// TIA Portal V16 export
// export: Created 2021-11-12T13:31:15.9471578Z, ExportSetting WithDefaults, DisplayName Totally Integrated Automation Portal, DisplayVersion V16 Update 3, DisplayName TIA Portal Version Control Interface, DisplayVersion V16 Update 2, DisplayName TIA Portal Openness, DisplayVersion V16 Update 3, DisplayName SINAMICS Startdrive Advanced, DisplayVersion V16 Update 5, DisplayName SINAMICS Startdrive G130, G150, S120, S150, SINAMICS MV, S210, DisplayVersion V16 Update 5, DisplayName SINAMICS Startdrive G110M, G120, G120C, G120D, G120P, G115D, DisplayVersion V16 Update 5, DisplayName STEP 7 Professional, DisplayVersion V16 Update 3, DisplayName STEP 7 Safety, DisplayVersion V16, DisplayName WinCC UA Professional, DisplayVersion V16 Update 3
FUNCTION_BLOCK "STD_RobotABB"   // FB1225, LAD
TITLE = STD_RobotABB
{ S7_Optimized_Access := 'TRUE' }
VERSION : 0.1
// Robot control
// stored: AutoNumber false, IsIECCheckEnabled false, IsRetainMemResEnabled false, MemoryReserve 100, SetENOAutomatically false, UDAEnableTagReadback false
   VAR_INPUT
      IS_ZoneM { ExternalAccessible := 'False'; ExternalVisible := 'False'; ExternalWritable := 'False'} : "UDT_Status_main";   // Main structure from zone
      IS_ZoneS { ExternalAccessible := 'False'; ExternalVisible := 'False'; ExternalWritable := 'False'} : "UDT_Zone_Status_specific";   // Specific structure from zone
      IS_Robot : "UDT_RobotABB_RobotDI";
      IS_Intl : "UDT_RobotABB_Interlock";
      IS_ZoneRel : "UDT_RobotABB_ZoneReleaseToRobot";
      IB1CtrlRun : Bool;   // Controller running in auto mode
      IB1LimSpd : Bool;   // Set robot maximal speed to safe speed (250mm/s default)
      IB1CnclJob : Bool;   // Cancel of robot job
      IB1StartJob : Bool;   // Start robot job - job number valid
      IB1AckEndOfJob : Bool;   // Acknowledge end of robot job
      IB1AlmSupp : Bool;   // Suppress alarms
      II_JobNr : UInt;   // Robot job number
      II_TypeNr : UInt;   // Robot type number
      II_PosNr : UInt;   // Robot position specification
   END_VAR
   VAR_OUTPUT
      OS_Status : Struct
         Main : "UDT_Status_main";
         Specific : "UDT_RobotABB_Status_specific";
         Error : "UDT_Error01";
      END_STRUCT;
      OS_Robot : "UDT_RobotABB_RobotDO";
   END_VAR
   VAR_IN_OUT
      XS_Parameter : "UDT_RobotABB_Parameter";
      XS_Command : "UDT_RobotABB_Command";
   END_VAR
   VAR
      SS_Alarm : Struct   // Device alarms
         RobotErr : Bool;   // Robot error - See teachpendant for further information
         Colsn : Bool;   // Motion supervision triggered
         JobNrNotMatch : Bool;   // Job number feedback does not match
         TypeNrNotMatch : Bool;   // Type number feedback does not match
         Res_0_4 : Bool;   // Reserve
         Res_0_5 : Bool;   // Reserve
         Res_0_6 : Bool;   // Reserve
         Res_0_7 : Bool;   // Reserve
      END_STRUCT;
      SS_Warning : Struct   // Device warnings
         LimSpd : Bool;   // Speed is limited to safe speed (250mm/s by default)
         NoTaskExec : Bool;   // Robot is not executing task
         NotOnPath : Bool;   // Robot is not on programmed path
         Res_0_3 : Bool;   // Reserve
         Res_0_4 : Bool;   // Reserve
         Res_0_5 : Bool;   // Reserve
         Res_0_6 : Bool;   // Reserve
         Res_0_7 : Bool;   // Reserve
      END_STRUCT;
      SS_RobotIn { S7_SetPoint := 'True'} : "UDT_RobotABB_RobotDI";
      SS_RobotOut { S7_SetPoint := 'True'} : "UDT_RobotABB_RobotDO";
      SS_SeqNr : UInt;
      SB1CollErr : Bool;   // Collective error from device
      SB1CollWrn : Bool;   // Collective warning from device
      SB1RobotReady : Bool;   // Robot ready to operation
      SB1StartJobReq : Bool;   // Start job request is detected
      SB1InitReq : Bool;   // Robot init request
      SB1InitTrg : Bool;   // Robot init request trigger
      SB1TrigPE1 : Bool;
      SB1TrigPE2 : Bool;
      SB1TrigPE3 : Bool;
      SB1CnclJobPE : Bool;
      SB1ServicePosReq : Bool;   // Request to go to/from service position
   END_VAR
   VAR_TEMP
      TS_Status : Struct
         Main : "UDT_Status_main";
         Specific : "UDT_RobotABB_Status_specific";
         Error : "UDT_Error01";
      END_STRUCT;
      TS_Parameter : "UDT_RobotABB_Parameter";
      TS_ZoneRel : Struct
         Zone : Array[0..#CI_StnNr] of Struct
            Allowed : Bool;
         END_STRUCT;
      END_STRUCT;
      TS_Intl : Struct
         Station : Array[0..#CI_StnNr] of Word;
      END_STRUCT;
      TS_Command : "UDT_RobotABB_Command";
      TW_StnIntlSpec : Word;
      "TW _StnIntlMask" : Word;   // Interlocks condition masked by request
      TW_StnIntlAckSpec : Word;   // Interlock conditions fulfilled PLC->Robot (selected station only)
      TI_StnIntlSpec : UInt;   // Interlock request Robot->PLC (Nr. of interlock in specific station)
      TI_IntStnNr : UInt;   // Interlock request Robot->PLC (station number)
      TI_RobotIntlAdj : UInt;   // Interlock number adjusted
      TI_InterlockLim : UInt;   // Interlock limitation
      TB1AckPulse : Bool;
      TB1AlmSupp : Bool;
      TI_RetVal : Int;
   END_VAR
   VAR CONSTANT
      CI_StnNr : UInt := 8;   // Number of stations used in Interfaces
   END_VAR
   VAR_TEMP   // added for the SCL form of the ladder/FBD networks
      _w1 : Bool;
      _w2 : Bool;
      _w3 : Bool;
      _w4 : Bool;
      _w5 : Bool;
   END_VAR
BEGIN

REGION Network 1: Clear temporary TS_Status - Main, Specific
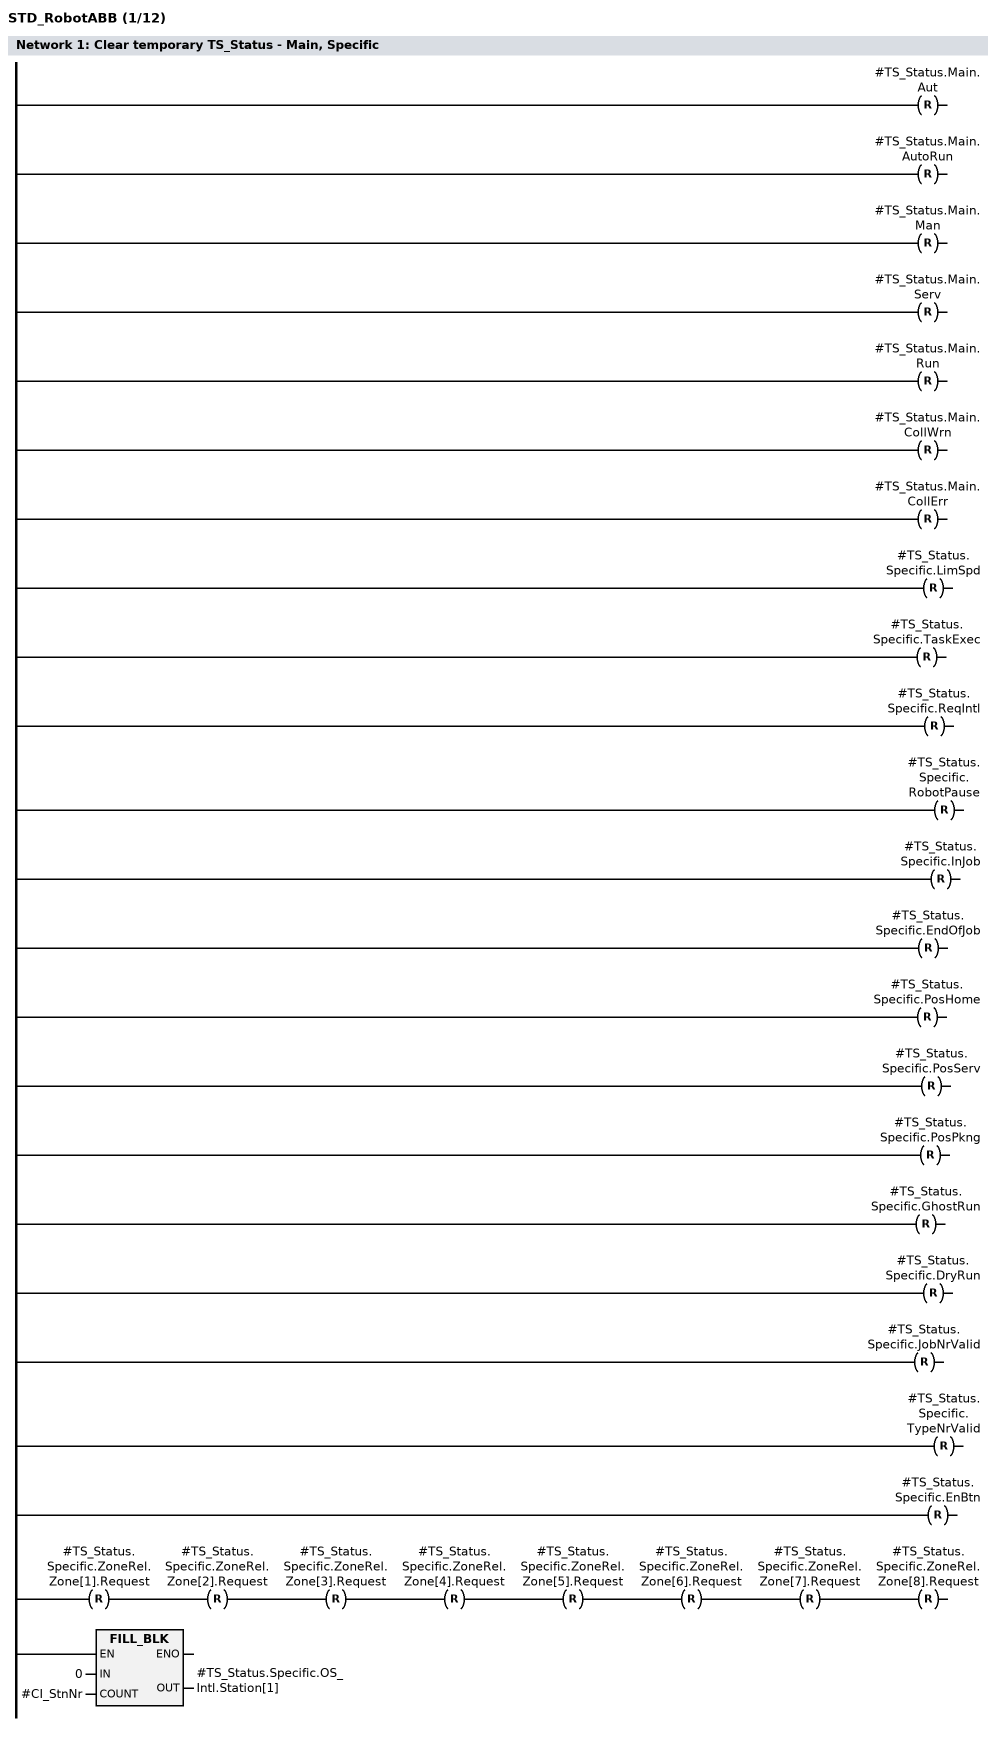
   RUNG wire#powerrail
      R_Coil( #TS_Status.Main.Aut )
   END_RUNG
   RUNG wire#powerrail
      R_Coil( #TS_Status.Main.AutoRun )
   END_RUNG
   RUNG wire#powerrail
      R_Coil( #TS_Status.Main.Man )
   END_RUNG
   RUNG wire#powerrail
      R_Coil( #TS_Status.Main.Serv )
   END_RUNG
   RUNG wire#powerrail
      R_Coil( #TS_Status.Main.Run )
   END_RUNG
   RUNG wire#powerrail
      R_Coil( #TS_Status.Main.CollWrn )
   END_RUNG
   RUNG wire#powerrail
      R_Coil( #TS_Status.Main.CollErr )
   END_RUNG
   RUNG wire#powerrail
      R_Coil( #TS_Status.Specific.LimSpd )
   END_RUNG
   RUNG wire#powerrail
      R_Coil( #TS_Status.Specific.TaskExec )
   END_RUNG
   RUNG wire#powerrail
      R_Coil( #TS_Status.Specific.ReqIntl )
   END_RUNG
   RUNG wire#powerrail
      R_Coil( #TS_Status.Specific.RobotPause )
   END_RUNG
   RUNG wire#powerrail
      R_Coil( #TS_Status.Specific.InJob )
   END_RUNG
   RUNG wire#powerrail
      R_Coil( #TS_Status.Specific.EndOfJob )
   END_RUNG
   RUNG wire#powerrail
      R_Coil( #TS_Status.Specific.PosHome )
   END_RUNG
   RUNG wire#powerrail
      R_Coil( #TS_Status.Specific.PosServ )
   END_RUNG
   RUNG wire#powerrail
      R_Coil( #TS_Status.Specific.PosPkng )
   END_RUNG
   RUNG wire#powerrail
      R_Coil( #TS_Status.Specific.GhostRun )
   END_RUNG
   RUNG wire#powerrail
      R_Coil( #TS_Status.Specific.DryRun )
   END_RUNG
   RUNG wire#powerrail
      R_Coil( #TS_Status.Specific.JobNrValid )
   END_RUNG
   RUNG wire#powerrail
      R_Coil( #TS_Status.Specific.TypeNrValid )
   END_RUNG
   RUNG wire#powerrail
      R_Coil( #TS_Status.Specific.EnBtn )
   END_RUNG
   RUNG wire#powerrail
      R_Coil( #TS_Status.Specific.ZoneRel.Zone[1].Request )
      R_Coil( #TS_Status.Specific.ZoneRel.Zone[2].Request )
      R_Coil( #TS_Status.Specific.ZoneRel.Zone[3].Request )
      R_Coil( #TS_Status.Specific.ZoneRel.Zone[4].Request )
      R_Coil( #TS_Status.Specific.ZoneRel.Zone[5].Request )
      R_Coil( #TS_Status.Specific.ZoneRel.Zone[6].Request )
      R_Coil( #TS_Status.Specific.ZoneRel.Zone[7].Request )
      R_Coil( #TS_Status.Specific.ZoneRel.Zone[8].Request )
   END_RUNG
   RUNG wire#powerrail
      { S7_GenerateENO := "TRUE" } FillBlockI(in := 0, count := #CI_StnNr, out => #TS_Status.Specific.OS_Intl.Station[1])
   END_RUNG
   // the same network as SCL:
   #TS_Status.Main.Aut := FALSE;
   #TS_Status.Main.AutoRun := FALSE;
   #TS_Status.Main.Man := FALSE;
   #TS_Status.Main.Serv := FALSE;
   #TS_Status.Main.Run := FALSE;
   #TS_Status.Main.CollWrn := FALSE;
   #TS_Status.Main.CollErr := FALSE;
   #TS_Status.Specific.LimSpd := FALSE;
   #TS_Status.Specific.TaskExec := FALSE;
   #TS_Status.Specific.ReqIntl := FALSE;
   #TS_Status.Specific.RobotPause := FALSE;
   #TS_Status.Specific.InJob := FALSE;
   #TS_Status.Specific.EndOfJob := FALSE;
   #TS_Status.Specific.PosHome := FALSE;
   #TS_Status.Specific.PosServ := FALSE;
   #TS_Status.Specific.PosPkng := FALSE;
   #TS_Status.Specific.GhostRun := FALSE;
   #TS_Status.Specific.DryRun := FALSE;
   #TS_Status.Specific.JobNrValid := FALSE;
   #TS_Status.Specific.TypeNrValid := FALSE;
   #TS_Status.Specific.EnBtn := FALSE;
   #TS_Status.Specific.ZoneRel.Zone[1].Request := FALSE;
   #TS_Status.Specific.ZoneRel.Zone[2].Request := FALSE;
   #TS_Status.Specific.ZoneRel.Zone[3].Request := FALSE;
   #TS_Status.Specific.ZoneRel.Zone[4].Request := FALSE;
   #TS_Status.Specific.ZoneRel.Zone[5].Request := FALSE;
   #TS_Status.Specific.ZoneRel.Zone[6].Request := FALSE;
   #TS_Status.Specific.ZoneRel.Zone[7].Request := FALSE;
   #TS_Status.Specific.ZoneRel.Zone[8].Request := FALSE;
   FILL_BLK(IN := 0, COUNT := #CI_StnNr, OUT => #TS_Status.Specific.OS_Intl.Station[1]);
END_REGION

REGION Network 2: Copy In/Out variables to temporary variables
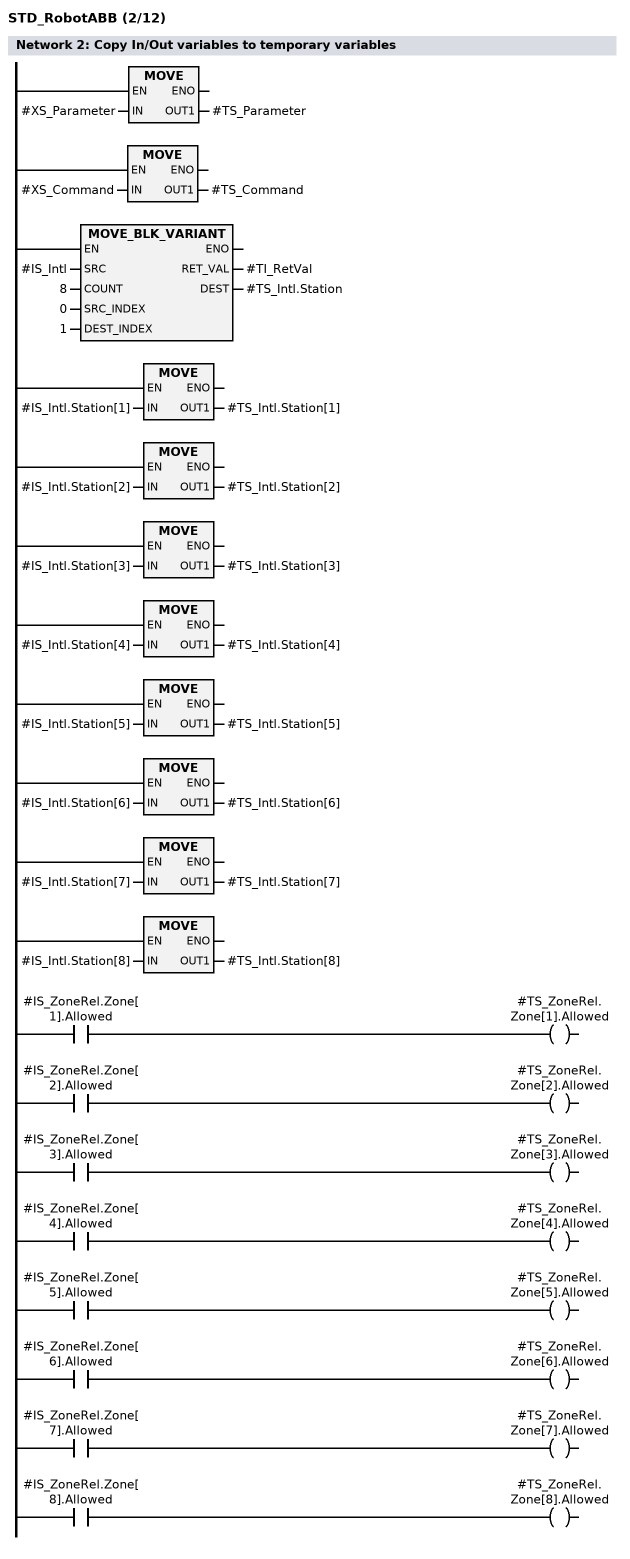
   RUNG wire#powerrail
      { S7_GenerateENO := "TRUE" } Move(in := #XS_Parameter, out1 => #TS_Parameter)
   END_RUNG
   RUNG wire#powerrail
      { S7_GenerateENO := "TRUE" } Move(in := #XS_Command, out1 => #TS_Command)
   END_RUNG
   RUNG wire#powerrail
      MOVE_BLK_VARIANT(SRC := #IS_Intl, COUNT := 8, SRC_INDEX := 0, DEST_INDEX := 1, Ret_Val => #TI_RetVal, DEST => #TS_Intl.Station)
   END_RUNG
   RUNG wire#powerrail
      Move(in := #IS_Intl.Station[1], out1 => #TS_Intl.Station[1])
   END_RUNG
   RUNG wire#powerrail
      Move(in := #IS_Intl.Station[2], out1 => #TS_Intl.Station[2])
   END_RUNG
   RUNG wire#powerrail
      Move(in := #IS_Intl.Station[3], out1 => #TS_Intl.Station[3])
   END_RUNG
   RUNG wire#powerrail
      Move(in := #IS_Intl.Station[4], out1 => #TS_Intl.Station[4])
   END_RUNG
   RUNG wire#powerrail
      Move(in := #IS_Intl.Station[5], out1 => #TS_Intl.Station[5])
   END_RUNG
   RUNG wire#powerrail
      Move(in := #IS_Intl.Station[6], out1 => #TS_Intl.Station[6])
   END_RUNG
   RUNG wire#powerrail
      Move(in := #IS_Intl.Station[7], out1 => #TS_Intl.Station[7])
   END_RUNG
   RUNG wire#powerrail
      Move(in := #IS_Intl.Station[8], out1 => #TS_Intl.Station[8])
   END_RUNG
   RUNG wire#powerrail
      Contact( #IS_ZoneRel.Zone[1].Allowed )
      Coil( #TS_ZoneRel.Zone[1].Allowed )
   END_RUNG
   RUNG wire#powerrail
      Contact( #IS_ZoneRel.Zone[2].Allowed )
      Coil( #TS_ZoneRel.Zone[2].Allowed )
   END_RUNG
   RUNG wire#powerrail
      Contact( #IS_ZoneRel.Zone[3].Allowed )
      Coil( #TS_ZoneRel.Zone[3].Allowed )
   END_RUNG
   RUNG wire#powerrail
      Contact( #IS_ZoneRel.Zone[4].Allowed )
      Coil( #TS_ZoneRel.Zone[4].Allowed )
   END_RUNG
   RUNG wire#powerrail
      Contact( #IS_ZoneRel.Zone[5].Allowed )
      Coil( #TS_ZoneRel.Zone[5].Allowed )
   END_RUNG
   RUNG wire#powerrail
      Contact( #IS_ZoneRel.Zone[6].Allowed )
      Coil( #TS_ZoneRel.Zone[6].Allowed )
   END_RUNG
   RUNG wire#powerrail
      Contact( #IS_ZoneRel.Zone[7].Allowed )
      Coil( #TS_ZoneRel.Zone[7].Allowed )
   END_RUNG
   RUNG wire#powerrail
      Contact( #IS_ZoneRel.Zone[8].Allowed )
      Coil( #TS_ZoneRel.Zone[8].Allowed )
   END_RUNG
   // the same network as SCL:
   #TS_Parameter := #XS_Parameter;
   #TS_Command := #XS_Command;
   #TI_RetVal := MOVE_BLK_VARIANT(SRC := #IS_Intl,
                           COUNT := 8,
                           SRC_INDEX := 0,
                           DEST_INDEX := 1,
                           DEST => #TS_Intl.Station);
   #TS_Intl.Station[1] := #IS_Intl.Station[1];
   #TS_Intl.Station[2] := #IS_Intl.Station[2];
   #TS_Intl.Station[3] := #IS_Intl.Station[3];
   #TS_Intl.Station[4] := #IS_Intl.Station[4];
   #TS_Intl.Station[5] := #IS_Intl.Station[5];
   #TS_Intl.Station[6] := #IS_Intl.Station[6];
   #TS_Intl.Station[7] := #IS_Intl.Station[7];
   #TS_Intl.Station[8] := #IS_Intl.Station[8];
   #TS_ZoneRel.Zone[1].Allowed := #IS_ZoneRel.Zone[1].Allowed;
   #TS_ZoneRel.Zone[2].Allowed := #IS_ZoneRel.Zone[2].Allowed;
   #TS_ZoneRel.Zone[3].Allowed := #IS_ZoneRel.Zone[3].Allowed;
   #TS_ZoneRel.Zone[4].Allowed := #IS_ZoneRel.Zone[4].Allowed;
   #TS_ZoneRel.Zone[5].Allowed := #IS_ZoneRel.Zone[5].Allowed;
   #TS_ZoneRel.Zone[6].Allowed := #IS_ZoneRel.Zone[6].Allowed;
   #TS_ZoneRel.Zone[7].Allowed := #IS_ZoneRel.Zone[7].Allowed;
   #TS_ZoneRel.Zone[8].Allowed := #IS_ZoneRel.Zone[8].Allowed;
END_REGION

REGION Network 3: Merge of alarm suppress
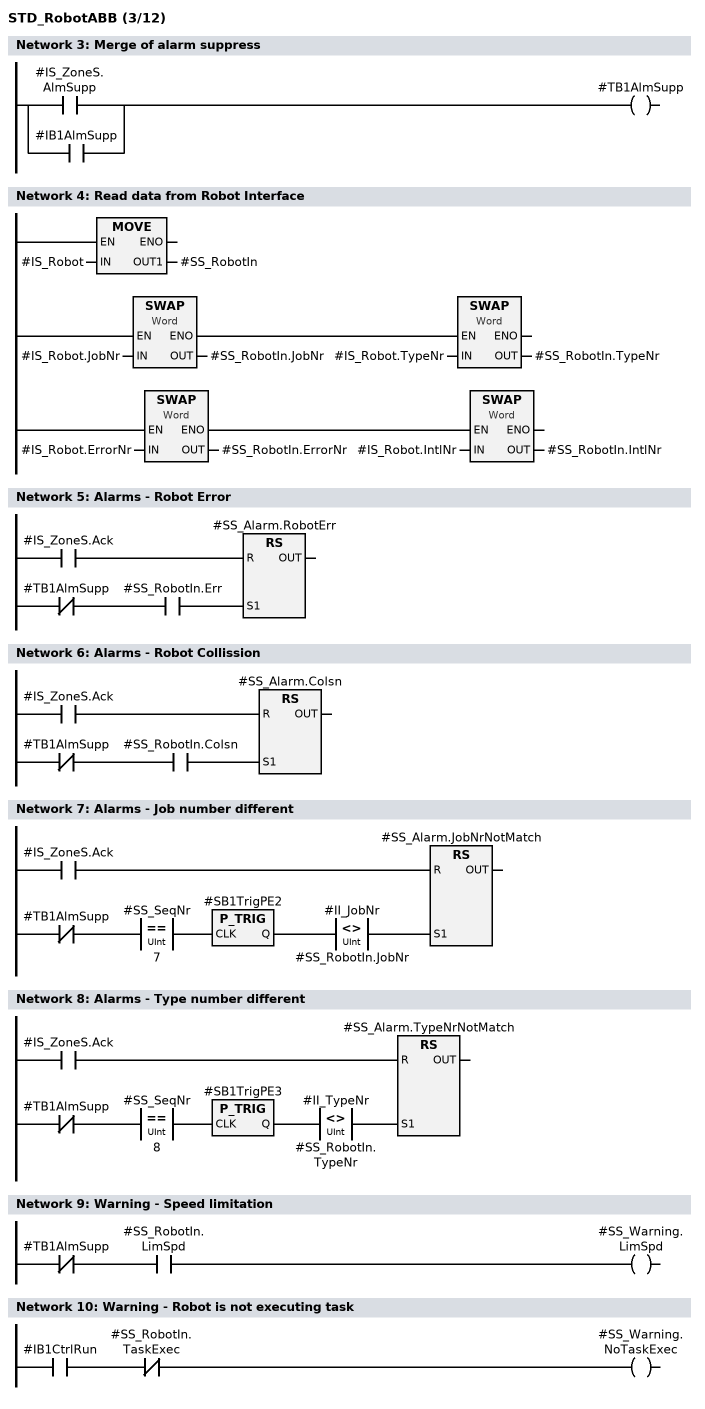
   RUNG wire#powerrail
      Contact( #IS_ZoneS.AlmSupp )
      wire#w1
      Coil( #TB1AlmSupp )
   END_RUNG
   RUNG wire#powerrail
      Contact( #IB1AlmSupp )
   END_RUNG wire#w1
   // the same network as SCL:
   #TB1AlmSupp := #IS_ZoneS.AlmSupp OR #IB1AlmSupp;
END_REGION

REGION Network 4: Read data from Robot Interface
   #SS_RobotIn := #IS_Robot;
   #SS_RobotIn.JobNr := SWAP(#IS_Robot.JobNr);
   #SS_RobotIn.TypeNr := SWAP(#IS_Robot.TypeNr);
   #SS_RobotIn.ErrorNr := SWAP(#IS_Robot.ErrorNr);
   #SS_RobotIn.IntlNr := SWAP(#IS_Robot.IntlNr);
END_REGION

REGION Network 5: Alarms - Robot Error
   RUNG wire#powerrail
      Contact( #IS_ZoneS.Ack )
      S_RS(operand := #SS_Alarm.RobotErr, s1 := wire#w1)
   END_RUNG
   RUNG wire#powerrail
      I_Contact( #TB1AlmSupp )
      Contact( #SS_RobotIn.Err )
   END_RUNG wire#w1
   // the same network as SCL:
   IF #IS_ZoneS.Ack THEN
       #SS_Alarm.RobotErr := FALSE;   // RS flip-flop
   END_IF;
   IF NOT #TB1AlmSupp AND #SS_RobotIn.Err THEN #SS_Alarm.RobotErr := TRUE; END_IF;
END_REGION

REGION Network 6: Alarms - Robot Collission
   RUNG wire#powerrail
      Contact( #IS_ZoneS.Ack )
      S_RS(operand := #SS_Alarm.Colsn, s1 := wire#w1)
   END_RUNG
   RUNG wire#powerrail
      I_Contact( #TB1AlmSupp )
      Contact( #SS_RobotIn.Colsn )
   END_RUNG wire#w1
   // the same network as SCL:
   IF #IS_ZoneS.Ack THEN
       #SS_Alarm.Colsn := FALSE;   // RS flip-flop
   END_IF;
   IF NOT #TB1AlmSupp AND #SS_RobotIn.Colsn THEN #SS_Alarm.Colsn := TRUE; END_IF;
END_REGION

REGION Network 7: Alarms - Job number different
   RUNG wire#powerrail
      Contact( #IS_ZoneS.Ack )
      S_RS(operand := #SS_Alarm.JobNrNotMatch, s1 := wire#w1)
   END_RUNG
   RUNG wire#powerrail
      I_Contact( #TB1AlmSupp )
      { S7_Templates := "SrcType := UInt" } EQ_Contact(in1 := #SS_SeqNr, in2 := 7)
      P_Trig( #SB1TrigPE2 )
      { S7_Templates := "SrcType := UInt" } NE_Contact(in1 := #II_JobNr, in2 := #SS_RobotIn.JobNr)
   END_RUNG wire#w1
   // the same network as SCL:
   #_w1 := NOT #TB1AlmSupp AND (#SS_SeqNr = 7);
   #_w2 := #_w1 AND NOT #SB1TrigPE2;   // rising edge
   #SB1TrigPE2 := #_w1;
   IF #IS_ZoneS.Ack THEN
       #SS_Alarm.JobNrNotMatch := FALSE;   // RS flip-flop
   END_IF;
   IF #_w2 AND (#II_JobNr <> #SS_RobotIn.JobNr) THEN #SS_Alarm.JobNrNotMatch := TRUE; END_IF;
END_REGION

REGION Network 8: Alarms - Type number different
   RUNG wire#powerrail
      Contact( #IS_ZoneS.Ack )
      S_RS(operand := #SS_Alarm.TypeNrNotMatch, s1 := wire#w1)
   END_RUNG
   RUNG wire#powerrail
      I_Contact( #TB1AlmSupp )
      { S7_Templates := "SrcType := UInt" } EQ_Contact(in1 := #SS_SeqNr, in2 := 8)
      P_Trig( #SB1TrigPE3 )
      { S7_Templates := "SrcType := UInt" } NE_Contact(in1 := #II_TypeNr, in2 := #SS_RobotIn.TypeNr)
   END_RUNG wire#w1
   // the same network as SCL:
   #_w1 := NOT #TB1AlmSupp AND (#SS_SeqNr = 8);
   #_w2 := #_w1 AND NOT #SB1TrigPE3;   // rising edge
   #SB1TrigPE3 := #_w1;
   IF #IS_ZoneS.Ack THEN
       #SS_Alarm.TypeNrNotMatch := FALSE;   // RS flip-flop
   END_IF;
   IF #_w2 AND (#II_TypeNr <> #SS_RobotIn.TypeNr) THEN #SS_Alarm.TypeNrNotMatch := TRUE; END_IF;
END_REGION

REGION Network 9: Warning - Speed limitation
   RUNG wire#powerrail
      I_Contact( #TB1AlmSupp )
      Contact( #SS_RobotIn.LimSpd )
      Coil( #SS_Warning.LimSpd )
   END_RUNG
   // the same network as SCL:
   #SS_Warning.LimSpd := NOT #TB1AlmSupp AND #SS_RobotIn.LimSpd;
END_REGION

REGION Network 10: Warning - Robot is not executing task
   RUNG wire#powerrail
      Contact( #IB1CtrlRun )
      I_Contact( #SS_RobotIn.TaskExec )
      Coil( #SS_Warning.NoTaskExec )
   END_RUNG
   // the same network as SCL:
   #SS_Warning.NoTaskExec := #IB1CtrlRun AND NOT #SS_RobotIn.TaskExec;
END_REGION

REGION Network 11: Warning - Robot is not programmed path
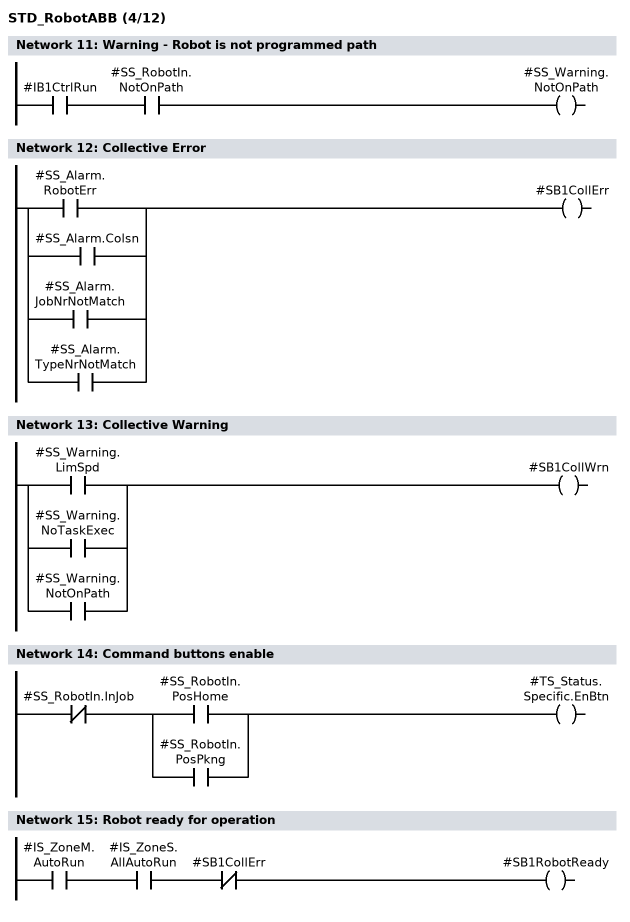
   RUNG wire#powerrail
      Contact( #IB1CtrlRun )
      Contact( #SS_RobotIn.NotOnPath )
      Coil( #SS_Warning.NotOnPath )
   END_RUNG
   // the same network as SCL:
   #SS_Warning.NotOnPath := #IB1CtrlRun AND #SS_RobotIn.NotOnPath;
END_REGION

REGION Network 12: Collective Error
   RUNG wire#powerrail
      Contact( #SS_Alarm.RobotErr )
      wire#w1
      Coil( #SB1CollErr )
   END_RUNG
   RUNG wire#powerrail
      Contact( #SS_Alarm.Colsn )
   END_RUNG wire#w1
   RUNG wire#powerrail
      Contact( #SS_Alarm.JobNrNotMatch )
   END_RUNG wire#w1
   RUNG wire#powerrail
      Contact( #SS_Alarm.TypeNrNotMatch )
   END_RUNG wire#w1
   // the same network as SCL:
   #SB1CollErr := #SS_Alarm.RobotErr OR #SS_Alarm.Colsn OR #SS_Alarm.JobNrNotMatch OR #SS_Alarm.TypeNrNotMatch;
END_REGION

REGION Network 13: Collective Warning
   RUNG wire#powerrail
      Contact( #SS_Warning.LimSpd )
      wire#w1
      Coil( #SB1CollWrn )
   END_RUNG
   RUNG wire#powerrail
      Contact( #SS_Warning.NoTaskExec )
   END_RUNG wire#w1
   RUNG wire#powerrail
      Contact( #SS_Warning.NotOnPath )
   END_RUNG wire#w1
   // the same network as SCL:
   #SB1CollWrn := #SS_Warning.LimSpd OR #SS_Warning.NoTaskExec OR #SS_Warning.NotOnPath;
END_REGION

REGION Network 14: Command buttons enable
   RUNG wire#powerrail
      I_Contact( #SS_RobotIn.InJob )
      wire#w1
      Contact( #SS_RobotIn.PosHome )
      wire#w2
      Coil( #TS_Status.Specific.EnBtn )
   END_RUNG
   RUNG wire#w1
      Contact( #SS_RobotIn.PosPkng )
   END_RUNG wire#w2
   // the same network as SCL:
   #TS_Status.Specific.EnBtn := NOT #SS_RobotIn.InJob AND (#SS_RobotIn.PosHome OR #SS_RobotIn.PosPkng);
END_REGION

REGION Network 15: Robot ready for operation
   RUNG wire#powerrail
      Contact( #IS_ZoneM.AutoRun )
      Contact( #IS_ZoneS.AllAutoRun )
      I_Contact( #SB1CollErr )
      Coil( #SB1RobotReady )
   END_RUNG
   // the same network as SCL:
   #SB1RobotReady := #IS_ZoneM.AutoRun AND #IS_ZoneS.AllAutoRun AND NOT #SB1CollErr;
END_REGION

REGION Network 16: Dry Run / Ghost Run
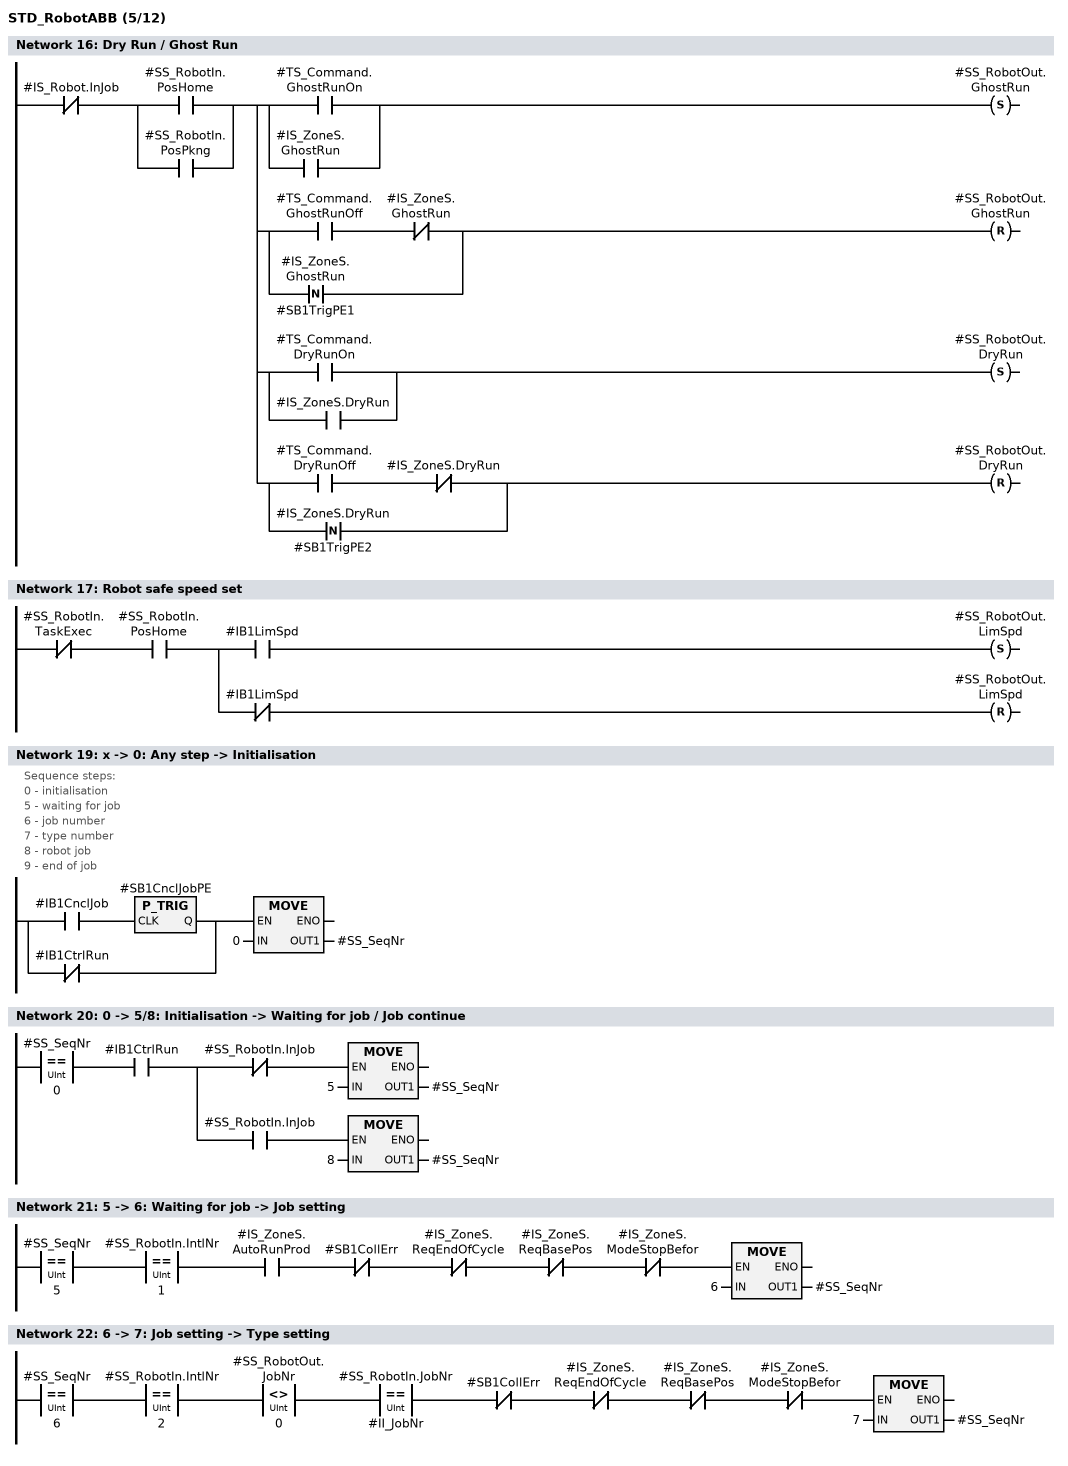
   RUNG wire#powerrail
      I_Contact( #IS_Robot.InJob )
      wire#w1
      Contact( #SS_RobotIn.PosHome )
      wire#w2
      Contact( #TS_Command.GhostRunOn )
      wire#w3
      S_Coil( #SS_RobotOut.GhostRun )
   END_RUNG
   RUNG wire#w1
      Contact( #SS_RobotIn.PosPkng )
   END_RUNG wire#w2
   RUNG wire#w2
      Contact( #IS_ZoneS.GhostRun )
   END_RUNG wire#w3
   RUNG wire#w2
      Contact( #TS_Command.GhostRunOff )
      I_Contact( #IS_ZoneS.GhostRun )
      wire#w4
      R_Coil( #SS_RobotOut.GhostRun )
   END_RUNG
   RUNG wire#w2
      N_Contact(operand := #IS_ZoneS.GhostRun, bit := #SB1TrigPE1)
   END_RUNG wire#w4
   RUNG wire#w2
      Contact( #TS_Command.DryRunOn )
      wire#w5
      S_Coil( #SS_RobotOut.DryRun )
   END_RUNG
   RUNG wire#w2
      Contact( #IS_ZoneS.DryRun )
   END_RUNG wire#w5
   RUNG wire#w2
      Contact( #TS_Command.DryRunOff )
      I_Contact( #IS_ZoneS.DryRun )
      wire#w6
      R_Coil( #SS_RobotOut.DryRun )
   END_RUNG
   RUNG wire#w2
      N_Contact(operand := #IS_ZoneS.DryRun, bit := #SB1TrigPE2)
   END_RUNG wire#w6
   // the same network as SCL:
   #_w1 := NOT #IS_Robot.InJob AND (#SS_RobotIn.PosHome OR #SS_RobotIn.PosPkng);
   IF #_w1 AND (#TS_Command.GhostRunOn OR #IS_ZoneS.GhostRun) THEN #SS_RobotOut.GhostRun := TRUE; END_IF;
   #_w2 := #_w1 AND NOT #IS_ZoneS.GhostRun AND #SB1TrigPE1;   // falling edge of #IS_ZoneS.GhostRun
   #SB1TrigPE1 := #IS_ZoneS.GhostRun;
   IF (#_w1 AND #TS_Command.GhostRunOff AND NOT #IS_ZoneS.GhostRun) OR #_w2 THEN
       #SS_RobotOut.GhostRun := FALSE;
   END_IF;
   IF #_w1 AND (#TS_Command.DryRunOn OR #IS_ZoneS.DryRun) THEN #SS_RobotOut.DryRun := TRUE; END_IF;
   #_w3 := #_w1 AND NOT #IS_ZoneS.DryRun AND #SB1TrigPE2;   // falling edge of #IS_ZoneS.DryRun
   #SB1TrigPE2 := #IS_ZoneS.DryRun;
   IF (#_w1 AND #TS_Command.DryRunOff AND NOT #IS_ZoneS.DryRun) OR #_w3 THEN
       #SS_RobotOut.DryRun := FALSE;
   END_IF;
END_REGION

REGION Network 17: Robot safe speed set
   RUNG wire#powerrail
      I_Contact( #SS_RobotIn.TaskExec )
      Contact( #SS_RobotIn.PosHome )
      wire#w1
      Contact( #IB1LimSpd )
      S_Coil( #SS_RobotOut.LimSpd )
   END_RUNG
   RUNG wire#w1
      I_Contact( #IB1LimSpd )
      R_Coil( #SS_RobotOut.LimSpd )
   END_RUNG
   // the same network as SCL:
   #_w1 := NOT #SS_RobotIn.TaskExec AND #SS_RobotIn.PosHome;
   IF #_w1 AND #IB1LimSpd THEN #SS_RobotOut.LimSpd := TRUE; END_IF;
   IF #_w1 AND NOT #IB1LimSpd THEN #SS_RobotOut.LimSpd := FALSE; END_IF;
END_REGION

REGION Network 18: *************** Robot control sequence - conditions ***************
END_REGION

REGION Network 19: x -> 0: Any step -> Initialisation
   // Sequence steps:
   // 0 - initialisation
   // 5 - waiting for job
   // 6 - job number
   // 7 - type number
   // 8 - robot job
   // 9 - end of job
   RUNG wire#powerrail
      Contact( #IB1CnclJob )
      P_Trig( #SB1CnclJobPE )
      wire#w1
      { S7_GenerateENO := "TRUE" } Move(in := 0, out1 => #SS_SeqNr)
   END_RUNG
   RUNG wire#powerrail
      I_Contact( #IB1CtrlRun )
   END_RUNG wire#w1
   // the same network as SCL:
   #_w1 := #IB1CnclJob AND NOT #SB1CnclJobPE;   // rising edge
   #SB1CnclJobPE := #IB1CnclJob;
   IF #_w1 OR NOT #IB1CtrlRun THEN #SS_SeqNr := 0; END_IF;
END_REGION

REGION Network 20: 0 -> 5/8: Initialisation -> Waiting for job / Job continue
   RUNG wire#powerrail
      { S7_Templates := "SrcType := UInt" } EQ_Contact(in1 := #SS_SeqNr, in2 := 0)
      Contact( #IB1CtrlRun )
      wire#w1
      I_Contact( #SS_RobotIn.InJob )
      { S7_GenerateENO := "TRUE" } Move(in := 5, out1 => #SS_SeqNr)
   END_RUNG
   RUNG wire#w1
      Contact( #SS_RobotIn.InJob )
      { S7_GenerateENO := "TRUE" } Move(in := 8, out1 => #SS_SeqNr)
   END_RUNG
   // the same network as SCL:
   #_w1 := (#SS_SeqNr = 0) AND #IB1CtrlRun;
   IF #_w1 AND NOT #SS_RobotIn.InJob THEN #SS_SeqNr := 5; END_IF;
   IF #_w1 AND #SS_RobotIn.InJob THEN #SS_SeqNr := 8; END_IF;
END_REGION

REGION Network 21: 5 -> 6: Waiting for job -> Job setting
   RUNG wire#powerrail
      { S7_Templates := "SrcType := UInt" } EQ_Contact(in1 := #SS_SeqNr, in2 := 5)
      { S7_Templates := "SrcType := UInt" } EQ_Contact(in1 := #SS_RobotIn.IntlNr, in2 := 1)
      Contact( #IS_ZoneS.AutoRunProd )
      I_Contact( #SB1CollErr )
      I_Contact( #IS_ZoneS.ReqEndOfCycle )
      I_Contact( #IS_ZoneS.ReqBasePos )
      I_Contact( #IS_ZoneS.ModeStopBefor )
      { S7_GenerateENO := "TRUE" } Move(in := 6, out1 => #SS_SeqNr)
   END_RUNG
   // the same network as SCL:
   IF (#SS_SeqNr = 5) AND (#SS_RobotIn.IntlNr = 1) AND #IS_ZoneS.AutoRunProd AND NOT #SB1CollErr AND NOT #IS_ZoneS.ReqEndOfCycle AND NOT #IS_ZoneS.ReqBasePos AND NOT #IS_ZoneS.ModeStopBefor THEN
       #SS_SeqNr := 6;
   END_IF;
END_REGION

REGION Network 22: 6 -> 7: Job setting -> Type setting
   RUNG wire#powerrail
      { S7_Templates := "SrcType := UInt" } EQ_Contact(in1 := #SS_SeqNr, in2 := 6)
      { S7_Templates := "SrcType := UInt" } EQ_Contact(in1 := #SS_RobotIn.IntlNr, in2 := 2)
      { S7_Templates := "SrcType := UInt" } NE_Contact(in1 := #SS_RobotOut.JobNr, in2 := 0)
      { S7_Templates := "SrcType := UInt" } EQ_Contact(in1 := #SS_RobotIn.JobNr, in2 := #II_JobNr)
      I_Contact( #SB1CollErr )
      I_Contact( #IS_ZoneS.ReqEndOfCycle )
      I_Contact( #IS_ZoneS.ReqBasePos )
      I_Contact( #IS_ZoneS.ModeStopBefor )
      { S7_GenerateENO := "TRUE" } Move(in := 7, out1 => #SS_SeqNr)
   END_RUNG
   // the same network as SCL:
   IF (#SS_SeqNr = 6) AND (#SS_RobotIn.IntlNr = 2) AND (#SS_RobotOut.JobNr <> 0) AND (#SS_RobotIn.JobNr = #II_JobNr) AND NOT #SB1CollErr AND NOT #IS_ZoneS.ReqEndOfCycle AND NOT #IS_ZoneS.ReqBasePos AND NOT #IS_ZoneS.ModeStopBefor THEN
       #SS_SeqNr := 7;
   END_IF;
END_REGION

REGION Network 23: 7 -> 8: Type setting -> Job active
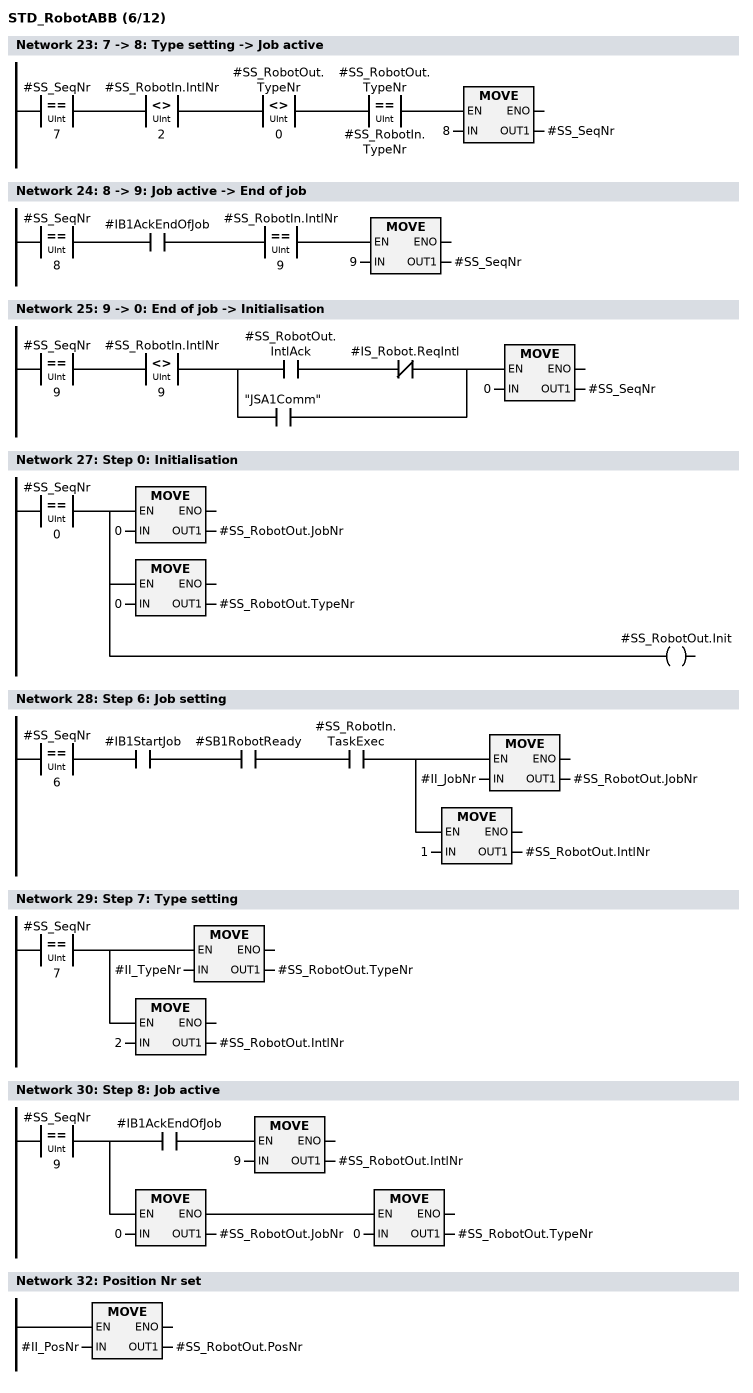
   RUNG wire#powerrail
      { S7_Templates := "SrcType := UInt" } EQ_Contact(in1 := #SS_SeqNr, in2 := 7)
      { S7_Templates := "SrcType := UInt" } NE_Contact(in1 := #SS_RobotIn.IntlNr, in2 := 2)
      { S7_Templates := "SrcType := UInt" } NE_Contact(in1 := #SS_RobotOut.TypeNr, in2 := 0)
      { S7_Templates := "SrcType := UInt" } EQ_Contact(in1 := #SS_RobotOut.TypeNr, in2 := #SS_RobotIn.TypeNr)
      { S7_GenerateENO := "TRUE" } Move(in := 8, out1 => #SS_SeqNr)
   END_RUNG
   // the same network as SCL:
   IF (#SS_SeqNr = 7) AND (#SS_RobotIn.IntlNr <> 2) AND (#SS_RobotOut.TypeNr <> 0) AND (#SS_RobotOut.TypeNr = #SS_RobotIn.TypeNr) THEN
       #SS_SeqNr := 8;
   END_IF;
END_REGION

REGION Network 24: 8 -> 9: Job active -> End of job
   RUNG wire#powerrail
      { S7_Templates := "SrcType := UInt" } EQ_Contact(in1 := #SS_SeqNr, in2 := 8)
      Contact( #IB1AckEndOfJob )
      { S7_Templates := "SrcType := UInt" } EQ_Contact(in1 := #SS_RobotIn.IntlNr, in2 := 9)
      { S7_GenerateENO := "TRUE" } Move(in := 9, out1 => #SS_SeqNr)
   END_RUNG
   // the same network as SCL:
   IF (#SS_SeqNr = 8) AND #IB1AckEndOfJob AND (#SS_RobotIn.IntlNr = 9) THEN #SS_SeqNr := 9; END_IF;
END_REGION

REGION Network 25: 9 -> 0: End of job -> Initialisation
   RUNG wire#powerrail
      { S7_Templates := "SrcType := UInt" } EQ_Contact(in1 := #SS_SeqNr, in2 := 9)
      { S7_Templates := "SrcType := UInt" } NE_Contact(in1 := #SS_RobotIn.IntlNr, in2 := 9)
      wire#w1
      Contact( #SS_RobotOut.IntlAck )
      I_Contact( #IS_Robot.ReqIntl )
      wire#w2
      { S7_GenerateENO := "TRUE" } Move(in := 0, out1 => #SS_SeqNr)
   END_RUNG
   RUNG wire#w1
      Contact( "JSA1Comm" )
   END_RUNG wire#w2
   // the same network as SCL:
   IF (#SS_SeqNr = 9) AND (#SS_RobotIn.IntlNr <> 9) AND ((#SS_RobotOut.IntlAck AND NOT #IS_Robot.ReqIntl) OR "JSA1Comm") THEN
       #SS_SeqNr := 0;
   END_IF;
END_REGION

REGION Network 26: *************** Robot control sequence - steps ***************
END_REGION

REGION Network 27: Step 0: Initialisation
   RUNG wire#powerrail
      { S7_Templates := "SrcType := UInt" } EQ_Contact(in1 := #SS_SeqNr, in2 := 0)
      wire#w1
      { S7_GenerateENO := "TRUE" } Move(in := 0, out1 => #SS_RobotOut.JobNr)
   END_RUNG
   RUNG wire#w1
      { S7_GenerateENO := "TRUE" } Move(in := 0, out1 => #SS_RobotOut.TypeNr)
   END_RUNG
   RUNG wire#w1
      Coil( #SS_RobotOut.Init )
   END_RUNG
   // the same network as SCL:
   #_w1 := #SS_SeqNr = 0;
   IF #_w1 THEN
       #SS_RobotOut.JobNr := 0;
       #SS_RobotOut.TypeNr := 0;
   END_IF;
   #SS_RobotOut.Init := #_w1;
END_REGION

REGION Network 28: Step 6: Job setting
   RUNG wire#powerrail
      { S7_Templates := "SrcType := UInt" } EQ_Contact(in1 := #SS_SeqNr, in2 := 6)
      Contact( #IB1StartJob )
      Contact( #SB1RobotReady )
      Contact( #SS_RobotIn.TaskExec )
      wire#w1
      { S7_GenerateENO := "TRUE" } Move(in := #II_JobNr, out1 => #SS_RobotOut.JobNr)
   END_RUNG
   RUNG wire#w1
      { S7_GenerateENO := "TRUE" } Move(in := 1, out1 => #SS_RobotOut.IntlNr)
   END_RUNG
   // the same network as SCL:
   IF (#SS_SeqNr = 6) AND #IB1StartJob AND #SB1RobotReady AND #SS_RobotIn.TaskExec THEN
       #SS_RobotOut.JobNr := #II_JobNr;
       #SS_RobotOut.IntlNr := 1;
   END_IF;
END_REGION

REGION Network 29: Step 7: Type setting
   RUNG wire#powerrail
      { S7_Templates := "SrcType := UInt" } EQ_Contact(in1 := #SS_SeqNr, in2 := 7)
      wire#w1
      { S7_GenerateENO := "TRUE" } Move(in := #II_TypeNr, out1 => #SS_RobotOut.TypeNr)
   END_RUNG
   RUNG wire#w1
      { S7_GenerateENO := "TRUE" } Move(in := 2, out1 => #SS_RobotOut.IntlNr)
   END_RUNG
   // the same network as SCL:
   IF #SS_SeqNr = 7 THEN
       #SS_RobotOut.TypeNr := #II_TypeNr;
       #SS_RobotOut.IntlNr := 2;
   END_IF;
END_REGION

REGION Network 30: Step 8: Job active
   RUNG wire#powerrail
      { S7_Templates := "SrcType := UInt" } EQ_Contact(in1 := #SS_SeqNr, in2 := 9)
      wire#w1
      Contact( #IB1AckEndOfJob )
      { S7_GenerateENO := "TRUE" } Move(in := 9, out1 => #SS_RobotOut.IntlNr)
   END_RUNG
   RUNG wire#w1
      { S7_GenerateENO := "TRUE" } Move(in := 0, out1 => #SS_RobotOut.JobNr)
      { S7_GenerateENO := "TRUE" } Move(in := 0, out1 => #SS_RobotOut.TypeNr)
   END_RUNG
   // the same network as SCL:
   // ENO of a box is taken as its EN; it also drops when the box reports an error
   #_w1 := #SS_SeqNr = 9;
   IF #_w1 AND #IB1AckEndOfJob THEN #SS_RobotOut.IntlNr := 9; END_IF;
   IF #_w1 THEN
       #SS_RobotOut.JobNr := 0;
       #SS_RobotOut.TypeNr := 0;
   END_IF;
END_REGION

REGION Network 31: *************** Robot control logic - Position Nr ***************
END_REGION

REGION Network 32: Position Nr set
   RUNG wire#powerrail
      Move(in := #II_PosNr, out1 => #SS_RobotOut.PosNr)
   END_RUNG
   // the same network as SCL:
   #SS_RobotOut.PosNr := #II_PosNr;
END_REGION

REGION Network 33: *************** Robot control logic - interlocs ***************
END_REGION

REGION Network 34: Interlock limitation
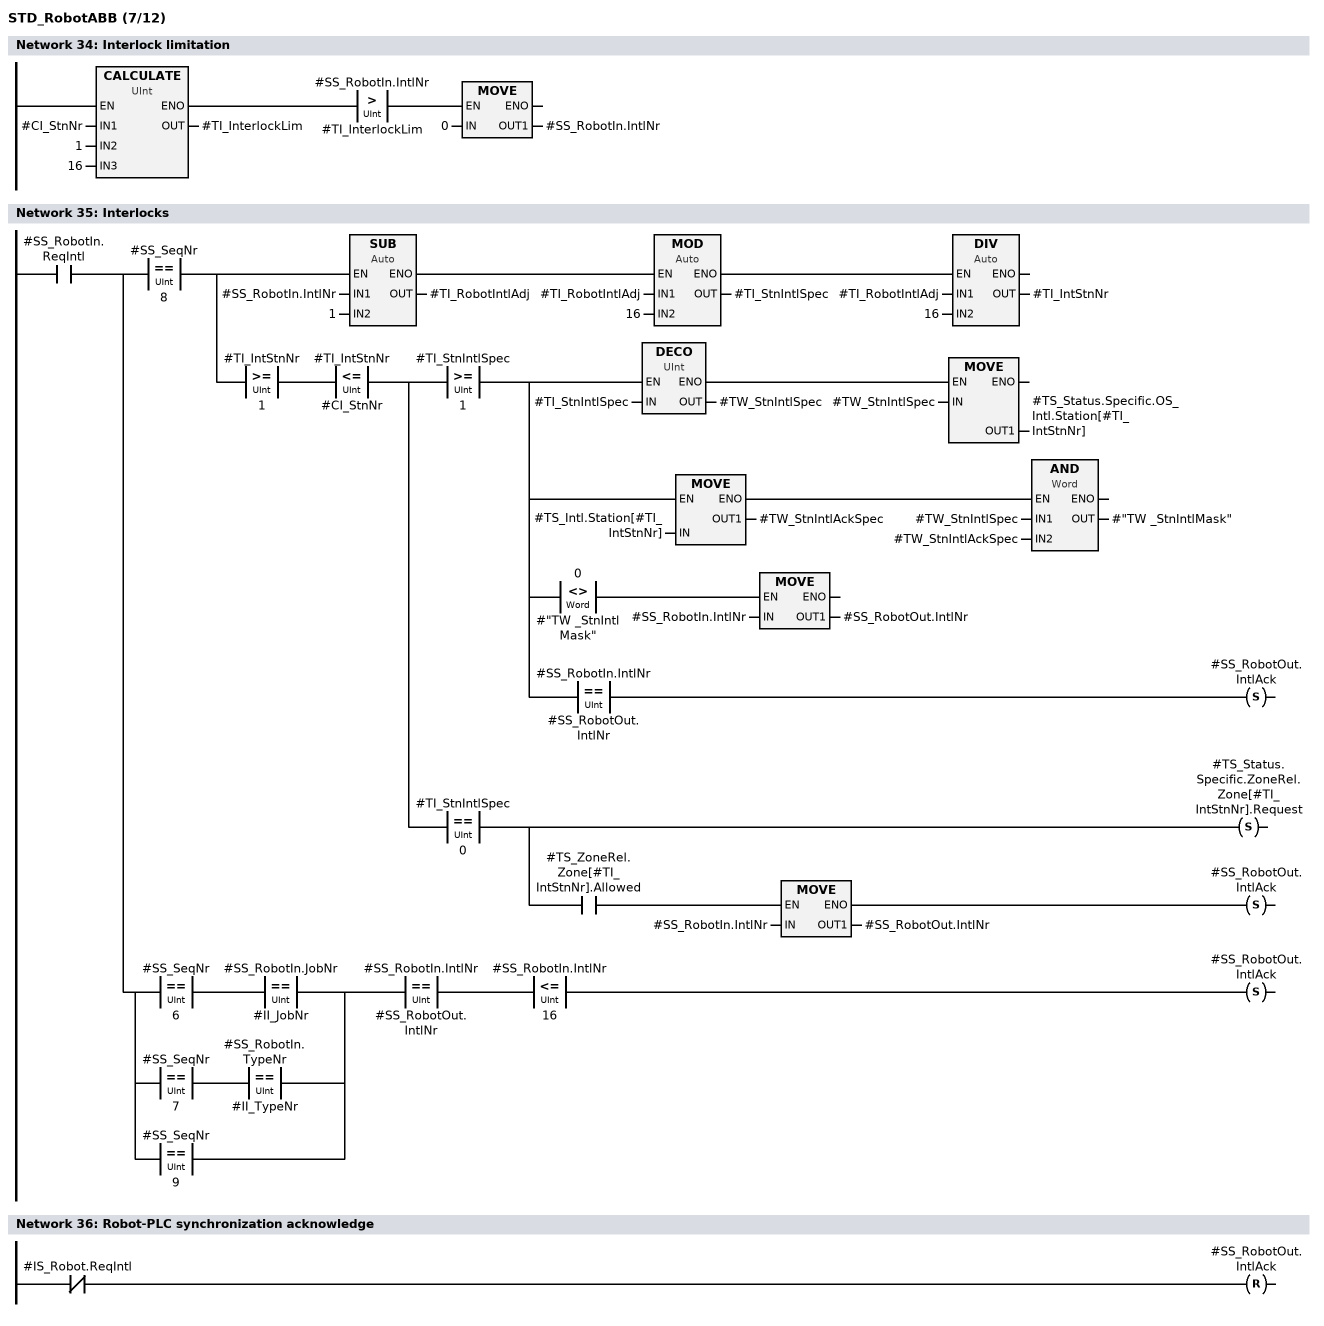
   RUNG wire#powerrail
      { S7_Templates := "SrcType := UInt"; S7_Expression := "((IN1+IN2)*IN3)" } Calculate(in1 := #CI_StnNr, in2 := 1, in3 := 16, out => #TI_InterlockLim)
      { S7_Templates := "SrcType := UInt" } GT_Contact(in1 := #SS_RobotIn.IntlNr, in2 := #TI_InterlockLim)
      Move(in := 0, out1 => #SS_RobotIn.IntlNr)
   END_RUNG
   // the same network as SCL:
   #TI_InterlockLim := ((#CI_StnNr+1)*16);
   IF #SS_RobotIn.IntlNr > #TI_InterlockLim THEN #SS_RobotIn.IntlNr := 0; END_IF;
END_REGION

REGION Network 35: Interlocks
   RUNG wire#powerrail
      Contact( #SS_RobotIn.ReqIntl )
      wire#w1
      { S7_Templates := "SrcType := UInt" } EQ_Contact(in1 := #SS_SeqNr, in2 := 8)
      wire#w2
      { S7_GenerateENO := "TRUE" } Sub(in1 := #SS_RobotIn.IntlNr, in2 := 1, out => #TI_RobotIntlAdj)
      { S7_GenerateENO := "TRUE" } Mod(in1 := #TI_RobotIntlAdj, in2 := 16, out => #TI_StnIntlSpec)
      { S7_GenerateENO := "TRUE" } Div(in1 := #TI_RobotIntlAdj, in2 := 16, out => #TI_IntStnNr)
   END_RUNG
   RUNG wire#w2
      { S7_Templates := "SrcType := UInt" } GE_Contact(in1 := #TI_IntStnNr, in2 := 1)
      { S7_Templates := "SrcType := UInt" } LE_Contact(in1 := #TI_IntStnNr, in2 := #CI_StnNr)
      wire#w3
      { S7_Templates := "SrcType := UInt" } GE_Contact(in1 := #TI_StnIntlSpec, in2 := 1)
      wire#w4
      { S7_Templates := "[value_type := UInt, return_type := Word]" } DECO(IN := #TI_StnIntlSpec, OUT => #TW_StnIntlSpec)
      { S7_GenerateENO := "TRUE" } Move(in := #TW_StnIntlSpec, out1 => #TS_Status.Specific.OS_Intl.Station[#TI_IntStnNr])
   END_RUNG
   RUNG wire#w4
      { S7_GenerateENO := "TRUE" } Move(in := #TS_Intl.Station[#TI_IntStnNr], out1 => #TW_StnIntlAckSpec)
      { S7_Templates := "SrcType := Word"; S7_GenerateENO := "TRUE" } And(in1 := #TW_StnIntlSpec, in2 := #TW_StnIntlAckSpec, out => #"TW _StnIntlMask")
   END_RUNG
   RUNG wire#w4
      { S7_Templates := "SrcType := Word" } NE_Contact(in1 := 0, in2 := #"TW _StnIntlMask")
      { S7_GenerateENO := "TRUE" } Move(in := #SS_RobotIn.IntlNr, out1 => #SS_RobotOut.IntlNr)
   END_RUNG
   RUNG wire#w4
      { S7_Templates := "SrcType := UInt" } EQ_Contact(in1 := #SS_RobotIn.IntlNr, in2 := #SS_RobotOut.IntlNr)
      S_Coil( #SS_RobotOut.IntlAck )
   END_RUNG
   RUNG wire#w3
      { S7_Templates := "SrcType := UInt" } EQ_Contact(in1 := #TI_StnIntlSpec, in2 := 0)
      wire#w5
      S_Coil( #TS_Status.Specific.ZoneRel.Zone[#TI_IntStnNr].Request )
   END_RUNG
   RUNG wire#w5
      Contact( #TS_ZoneRel.Zone[#TI_IntStnNr].Allowed )
      { S7_GenerateENO := "TRUE" } Move(in := #SS_RobotIn.IntlNr, out1 => #SS_RobotOut.IntlNr)
      S_Coil( #SS_RobotOut.IntlAck )
   END_RUNG
   RUNG wire#w1
      { S7_Templates := "SrcType := UInt" } EQ_Contact(in1 := #SS_SeqNr, in2 := 6)
      { S7_Templates := "SrcType := UInt" } EQ_Contact(in1 := #SS_RobotIn.JobNr, in2 := #II_JobNr)
      wire#w6
      { S7_Templates := "SrcType := UInt" } EQ_Contact(in1 := #SS_RobotIn.IntlNr, in2 := #SS_RobotOut.IntlNr)
      { S7_Templates := "SrcType := UInt" } LE_Contact(in1 := #SS_RobotIn.IntlNr, in2 := 16)
      S_Coil( #SS_RobotOut.IntlAck )
   END_RUNG
   RUNG wire#w1
      { S7_Templates := "SrcType := UInt" } EQ_Contact(in1 := #SS_SeqNr, in2 := 7)
      { S7_Templates := "SrcType := UInt" } EQ_Contact(in1 := #SS_RobotIn.TypeNr, in2 := #II_TypeNr)
   END_RUNG wire#w6
   RUNG wire#w1
      { S7_Templates := "SrcType := UInt" } EQ_Contact(in1 := #SS_SeqNr, in2 := 9)
   END_RUNG wire#w6
   // the same network as SCL:
   // ENO of a box is taken as its EN; it also drops when the box reports an error
   #_w1 := #SS_RobotIn.ReqIntl AND (#SS_SeqNr = 8);
   IF #_w1 THEN
       #TI_RobotIntlAdj := #SS_RobotIn.IntlNr - 1;
       #TI_StnIntlSpec := #TI_RobotIntlAdj MOD 16;
       #TI_IntStnNr := #TI_RobotIntlAdj / 16;
   END_IF;
   #_w2 := #_w1 AND (#TI_IntStnNr >= 1) AND (#TI_IntStnNr <= #CI_StnNr);
   #_w3 := #_w2 AND (#TI_StnIntlSpec >= 1);
   DECO(EN := #_w3, IN := #TI_StnIntlSpec, OUT => #TW_StnIntlSpec, ENO => #_w4);
   IF #_w4 THEN #TS_Status.Specific.OS_Intl.Station[#TI_IntStnNr] := #TW_StnIntlSpec; END_IF;
   IF #_w3 THEN
       #TW_StnIntlAckSpec := #TS_Intl.Station[#TI_IntStnNr];
       #"TW _StnIntlMask" := #TW_StnIntlSpec AND #TW_StnIntlAckSpec;
   END_IF;
   IF #_w3 AND (0 <> #"TW _StnIntlMask") THEN #SS_RobotOut.IntlNr := #SS_RobotIn.IntlNr; END_IF;
   IF #_w3 AND (#SS_RobotIn.IntlNr = #SS_RobotOut.IntlNr) THEN #SS_RobotOut.IntlAck := TRUE; END_IF;
   #_w5 := #_w2 AND (#TI_StnIntlSpec = 0);
   IF #_w5 THEN #TS_Status.Specific.ZoneRel.Zone[#TI_IntStnNr].Request := TRUE; END_IF;
   IF #_w5 AND #TS_ZoneRel.Zone[#TI_IntStnNr].Allowed THEN
       #SS_RobotOut.IntlNr := #SS_RobotIn.IntlNr;
       #SS_RobotOut.IntlAck := TRUE;
   END_IF;
   IF #SS_RobotIn.ReqIntl AND (((#SS_SeqNr = 6) AND (#SS_RobotIn.JobNr = #II_JobNr)) OR ((#SS_SeqNr = 7) AND (#SS_RobotIn.TypeNr = #II_TypeNr)) OR (#SS_SeqNr = 9)) AND (#SS_RobotIn.IntlNr = #SS_RobotOut.IntlNr) AND (#SS_RobotIn.IntlNr <= 16) THEN
       #SS_RobotOut.IntlAck := TRUE;
   END_IF;
END_REGION

REGION Network 36: Robot-PLC synchronization acknowledge
   RUNG wire#powerrail
      I_Contact( #IS_Robot.ReqIntl )
      R_Coil( #SS_RobotOut.IntlAck )
   END_RUNG
   // the same network as SCL:
   IF NOT #IS_Robot.ReqIntl THEN #SS_RobotOut.IntlAck := FALSE; END_IF;
END_REGION

REGION Network 37: *************** Other logic ***************
END_REGION

REGION Network 38: Filling the Main status
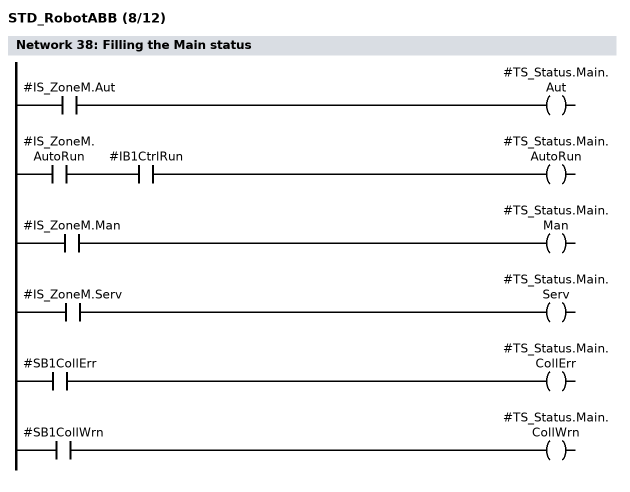
   RUNG wire#powerrail
      Contact( #IS_ZoneM.Aut )
      Coil( #TS_Status.Main.Aut )
   END_RUNG
   RUNG wire#powerrail
      Contact( #IS_ZoneM.AutoRun )
      Contact( #IB1CtrlRun )
      Coil( #TS_Status.Main.AutoRun )
   END_RUNG
   RUNG wire#powerrail
      Contact( #IS_ZoneM.Man )
      Coil( #TS_Status.Main.Man )
   END_RUNG
   RUNG wire#powerrail
      Contact( #IS_ZoneM.Serv )
      Coil( #TS_Status.Main.Serv )
   END_RUNG
   RUNG wire#powerrail
      Contact( #SB1CollErr )
      Coil( #TS_Status.Main.CollErr )
   END_RUNG
   RUNG wire#powerrail
      Contact( #SB1CollWrn )
      Coil( #TS_Status.Main.CollWrn )
   END_RUNG
   // the same network as SCL:
   #TS_Status.Main.Aut := #IS_ZoneM.Aut;
   #TS_Status.Main.AutoRun := #IS_ZoneM.AutoRun AND #IB1CtrlRun;
   #TS_Status.Main.Man := #IS_ZoneM.Man;
   #TS_Status.Main.Serv := #IS_ZoneM.Serv;
   #TS_Status.Main.CollErr := #SB1CollErr;
   #TS_Status.Main.CollWrn := #SB1CollWrn;
END_REGION

REGION Network 39: Status Specific
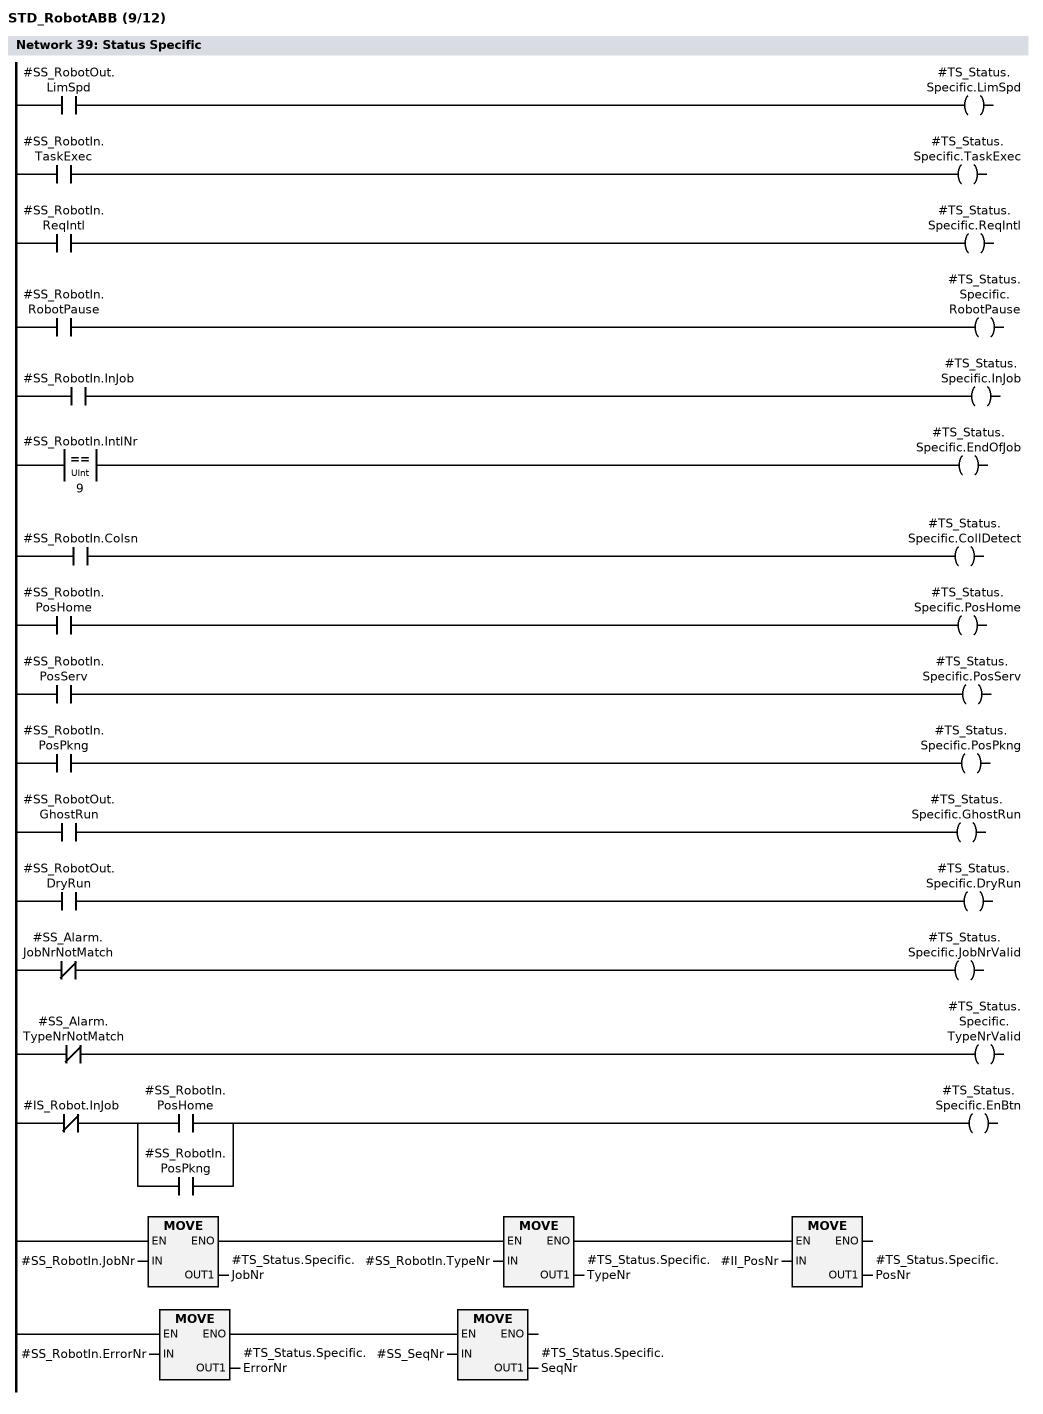
   RUNG wire#powerrail
      Contact( #SS_RobotOut.LimSpd )
      Coil( #TS_Status.Specific.LimSpd )
   END_RUNG
   RUNG wire#powerrail
      Contact( #SS_RobotIn.TaskExec )
      Coil( #TS_Status.Specific.TaskExec )
   END_RUNG
   RUNG wire#powerrail
      Contact( #SS_RobotIn.ReqIntl )
      Coil( #TS_Status.Specific.ReqIntl )
   END_RUNG
   RUNG wire#powerrail
      Contact( #SS_RobotIn.RobotPause )
      Coil( #TS_Status.Specific.RobotPause )
   END_RUNG
   RUNG wire#powerrail
      Contact( #SS_RobotIn.InJob )
      Coil( #TS_Status.Specific.InJob )
   END_RUNG
   RUNG wire#powerrail
      { S7_Templates := "SrcType := UInt" } EQ_Contact(in1 := #SS_RobotIn.IntlNr, in2 := 9)
      Coil( #TS_Status.Specific.EndOfJob )
   END_RUNG
   RUNG wire#powerrail
      Contact( #SS_RobotIn.Colsn )
      Coil( #TS_Status.Specific.CollDetect )
   END_RUNG
   RUNG wire#powerrail
      Contact( #SS_RobotIn.PosHome )
      Coil( #TS_Status.Specific.PosHome )
   END_RUNG
   RUNG wire#powerrail
      Contact( #SS_RobotIn.PosServ )
      Coil( #TS_Status.Specific.PosServ )
   END_RUNG
   RUNG wire#powerrail
      Contact( #SS_RobotIn.PosPkng )
      Coil( #TS_Status.Specific.PosPkng )
   END_RUNG
   RUNG wire#powerrail
      Contact( #SS_RobotOut.GhostRun )
      Coil( #TS_Status.Specific.GhostRun )
   END_RUNG
   RUNG wire#powerrail
      Contact( #SS_RobotOut.DryRun )
      Coil( #TS_Status.Specific.DryRun )
   END_RUNG
   RUNG wire#powerrail
      I_Contact( #SS_Alarm.JobNrNotMatch )
      Coil( #TS_Status.Specific.JobNrValid )
   END_RUNG
   RUNG wire#powerrail
      I_Contact( #SS_Alarm.TypeNrNotMatch )
      Coil( #TS_Status.Specific.TypeNrValid )
   END_RUNG
   RUNG wire#powerrail
      I_Contact( #IS_Robot.InJob )
      wire#w1
      Contact( #SS_RobotIn.PosHome )
      wire#w2
      Coil( #TS_Status.Specific.EnBtn )
   END_RUNG
   RUNG wire#w1
      Contact( #SS_RobotIn.PosPkng )
   END_RUNG wire#w2
   RUNG wire#powerrail
      { S7_GenerateENO := "TRUE" } Move(in := #SS_RobotIn.JobNr, out1 => #TS_Status.Specific.JobNr)
      { S7_GenerateENO := "TRUE" } Move(in := #SS_RobotIn.TypeNr, out1 => #TS_Status.Specific.TypeNr)
      { S7_GenerateENO := "TRUE" } Move(in := #II_PosNr, out1 => #TS_Status.Specific.PosNr)
   END_RUNG
   RUNG wire#powerrail
      { S7_GenerateENO := "TRUE" } Move(in := #SS_RobotIn.ErrorNr, out1 => #TS_Status.Specific.ErrorNr)
      { S7_GenerateENO := "TRUE" } Move(in := #SS_SeqNr, out1 => #TS_Status.Specific.SeqNr)
   END_RUNG
   // the same network as SCL:
   // ENO of a box is taken as its EN; it also drops when the box reports an error
   #TS_Status.Specific.LimSpd := #SS_RobotOut.LimSpd;
   #TS_Status.Specific.TaskExec := #SS_RobotIn.TaskExec;
   #TS_Status.Specific.ReqIntl := #SS_RobotIn.ReqIntl;
   #TS_Status.Specific.RobotPause := #SS_RobotIn.RobotPause;
   #TS_Status.Specific.InJob := #SS_RobotIn.InJob;
   #TS_Status.Specific.EndOfJob := #SS_RobotIn.IntlNr = 9;
   #TS_Status.Specific.CollDetect := #SS_RobotIn.Colsn;
   #TS_Status.Specific.PosHome := #SS_RobotIn.PosHome;
   #TS_Status.Specific.PosServ := #SS_RobotIn.PosServ;
   #TS_Status.Specific.PosPkng := #SS_RobotIn.PosPkng;
   #TS_Status.Specific.GhostRun := #SS_RobotOut.GhostRun;
   #TS_Status.Specific.DryRun := #SS_RobotOut.DryRun;
   #TS_Status.Specific.JobNrValid := NOT #SS_Alarm.JobNrNotMatch;
   #TS_Status.Specific.TypeNrValid := NOT #SS_Alarm.TypeNrNotMatch;
   #TS_Status.Specific.EnBtn := NOT #IS_Robot.InJob AND (#SS_RobotIn.PosHome OR #SS_RobotIn.PosPkng);
   #TS_Status.Specific.JobNr := #SS_RobotIn.JobNr;
   #TS_Status.Specific.TypeNr := #SS_RobotIn.TypeNr;
   #TS_Status.Specific.PosNr := #II_PosNr;
   #TS_Status.Specific.ErrorNr := #SS_RobotIn.ErrorNr;
   #TS_Status.Specific.SeqNr := #SS_SeqNr;
END_REGION

REGION Network 40: Station Release
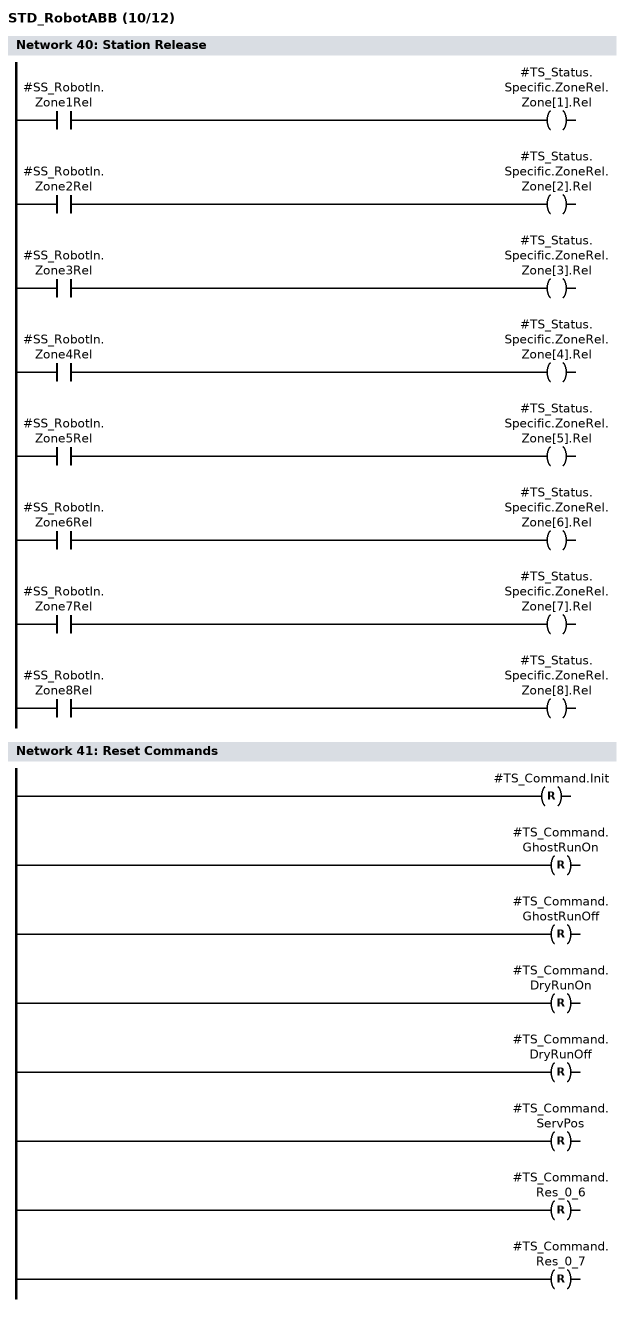
   RUNG wire#powerrail
      Contact( #SS_RobotIn.Zone1Rel )
      Coil( #TS_Status.Specific.ZoneRel.Zone[1].Rel )
   END_RUNG
   RUNG wire#powerrail
      Contact( #SS_RobotIn.Zone2Rel )
      Coil( #TS_Status.Specific.ZoneRel.Zone[2].Rel )
   END_RUNG
   RUNG wire#powerrail
      Contact( #SS_RobotIn.Zone3Rel )
      Coil( #TS_Status.Specific.ZoneRel.Zone[3].Rel )
   END_RUNG
   RUNG wire#powerrail
      Contact( #SS_RobotIn.Zone4Rel )
      Coil( #TS_Status.Specific.ZoneRel.Zone[4].Rel )
   END_RUNG
   RUNG wire#powerrail
      Contact( #SS_RobotIn.Zone5Rel )
      Coil( #TS_Status.Specific.ZoneRel.Zone[5].Rel )
   END_RUNG
   RUNG wire#powerrail
      Contact( #SS_RobotIn.Zone6Rel )
      Coil( #TS_Status.Specific.ZoneRel.Zone[6].Rel )
   END_RUNG
   RUNG wire#powerrail
      Contact( #SS_RobotIn.Zone7Rel )
      Coil( #TS_Status.Specific.ZoneRel.Zone[7].Rel )
   END_RUNG
   RUNG wire#powerrail
      Contact( #SS_RobotIn.Zone8Rel )
      Coil( #TS_Status.Specific.ZoneRel.Zone[8].Rel )
   END_RUNG
   // the same network as SCL:
   #TS_Status.Specific.ZoneRel.Zone[1].Rel := #SS_RobotIn.Zone1Rel;
   #TS_Status.Specific.ZoneRel.Zone[2].Rel := #SS_RobotIn.Zone2Rel;
   #TS_Status.Specific.ZoneRel.Zone[3].Rel := #SS_RobotIn.Zone3Rel;
   #TS_Status.Specific.ZoneRel.Zone[4].Rel := #SS_RobotIn.Zone4Rel;
   #TS_Status.Specific.ZoneRel.Zone[5].Rel := #SS_RobotIn.Zone5Rel;
   #TS_Status.Specific.ZoneRel.Zone[6].Rel := #SS_RobotIn.Zone6Rel;
   #TS_Status.Specific.ZoneRel.Zone[7].Rel := #SS_RobotIn.Zone7Rel;
   #TS_Status.Specific.ZoneRel.Zone[8].Rel := #SS_RobotIn.Zone8Rel;
END_REGION

REGION Network 41: Reset Commands
   RUNG wire#powerrail
      R_Coil( #TS_Command.Init )
   END_RUNG
   RUNG wire#powerrail
      R_Coil( #TS_Command.GhostRunOn )
   END_RUNG
   RUNG wire#powerrail
      R_Coil( #TS_Command.GhostRunOff )
   END_RUNG
   RUNG wire#powerrail
      R_Coil( #TS_Command.DryRunOn )
   END_RUNG
   RUNG wire#powerrail
      R_Coil( #TS_Command.DryRunOff )
   END_RUNG
   RUNG wire#powerrail
      R_Coil( #TS_Command.ServPos )
   END_RUNG
   RUNG wire#powerrail
      R_Coil( #TS_Command.Res_0_6 )
   END_RUNG
   RUNG wire#powerrail
      R_Coil( #TS_Command.Res_0_7 )
   END_RUNG
   // the same network as SCL:
   #TS_Command.Init := FALSE;
   #TS_Command.GhostRunOn := FALSE;
   #TS_Command.GhostRunOff := FALSE;
   #TS_Command.DryRunOn := FALSE;
   #TS_Command.DryRunOff := FALSE;
   #TS_Command.ServPos := FALSE;
   #TS_Command.Res_0_6 := FALSE;
   #TS_Command.Res_0_7 := FALSE;
END_REGION

REGION Network 42: Alarms - copy to output structure
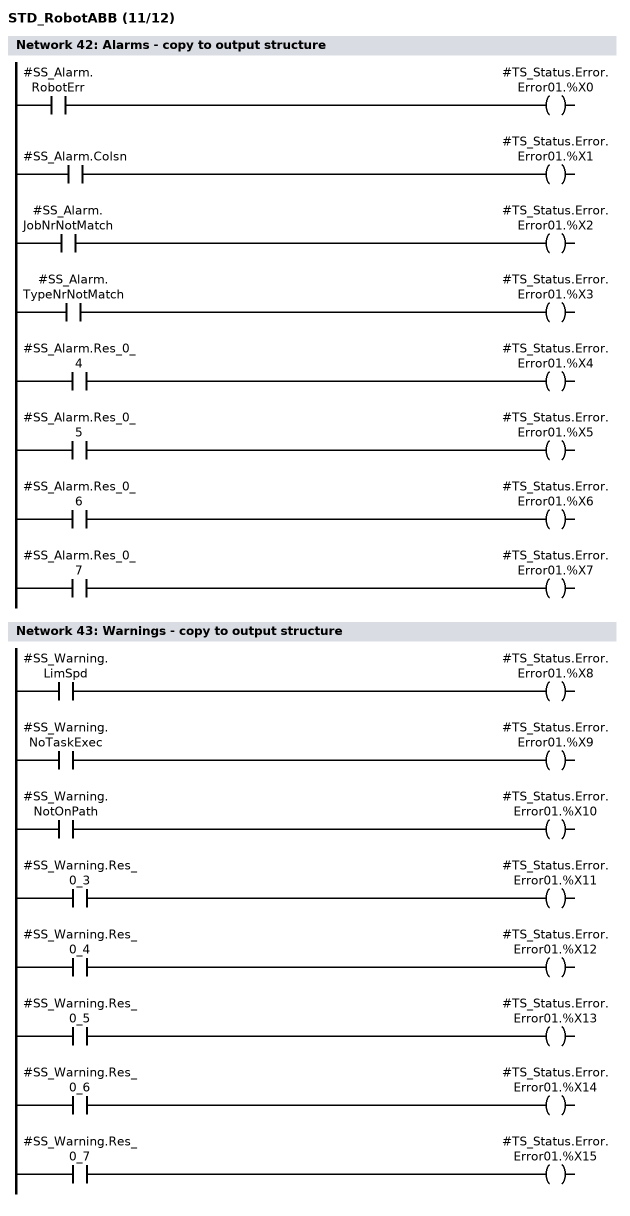
   RUNG wire#powerrail
      Contact( #SS_Alarm.RobotErr )
      Coil( #TS_Status.Error.Error01.%X0 )
   END_RUNG
   RUNG wire#powerrail
      Contact( #SS_Alarm.Colsn )
      Coil( #TS_Status.Error.Error01.%X1 )
   END_RUNG
   RUNG wire#powerrail
      Contact( #SS_Alarm.JobNrNotMatch )
      Coil( #TS_Status.Error.Error01.%X2 )
   END_RUNG
   RUNG wire#powerrail
      Contact( #SS_Alarm.TypeNrNotMatch )
      Coil( #TS_Status.Error.Error01.%X3 )
   END_RUNG
   RUNG wire#powerrail
      Contact( #SS_Alarm.Res_0_4 )
      Coil( #TS_Status.Error.Error01.%X4 )
   END_RUNG
   RUNG wire#powerrail
      Contact( #SS_Alarm.Res_0_5 )
      Coil( #TS_Status.Error.Error01.%X5 )
   END_RUNG
   RUNG wire#powerrail
      Contact( #SS_Alarm.Res_0_6 )
      Coil( #TS_Status.Error.Error01.%X6 )
   END_RUNG
   RUNG wire#powerrail
      Contact( #SS_Alarm.Res_0_7 )
      Coil( #TS_Status.Error.Error01.%X7 )
   END_RUNG
   // the same network as SCL:
   #TS_Status.Error.Error01.%X0 := #SS_Alarm.RobotErr;
   #TS_Status.Error.Error01.%X1 := #SS_Alarm.Colsn;
   #TS_Status.Error.Error01.%X2 := #SS_Alarm.JobNrNotMatch;
   #TS_Status.Error.Error01.%X3 := #SS_Alarm.TypeNrNotMatch;
   #TS_Status.Error.Error01.%X4 := #SS_Alarm.Res_0_4;
   #TS_Status.Error.Error01.%X5 := #SS_Alarm.Res_0_5;
   #TS_Status.Error.Error01.%X6 := #SS_Alarm.Res_0_6;
   #TS_Status.Error.Error01.%X7 := #SS_Alarm.Res_0_7;
END_REGION

REGION Network 43: Warnings - copy to output structure
   RUNG wire#powerrail
      Contact( #SS_Warning.LimSpd )
      Coil( #TS_Status.Error.Error01.%X8 )
   END_RUNG
   RUNG wire#powerrail
      Contact( #SS_Warning.NoTaskExec )
      Coil( #TS_Status.Error.Error01.%X9 )
   END_RUNG
   RUNG wire#powerrail
      Contact( #SS_Warning.NotOnPath )
      Coil( #TS_Status.Error.Error01.%X10 )
   END_RUNG
   RUNG wire#powerrail
      Contact( #SS_Warning.Res_0_3 )
      Coil( #TS_Status.Error.Error01.%X11 )
   END_RUNG
   RUNG wire#powerrail
      Contact( #SS_Warning.Res_0_4 )
      Coil( #TS_Status.Error.Error01.%X12 )
   END_RUNG
   RUNG wire#powerrail
      Contact( #SS_Warning.Res_0_5 )
      Coil( #TS_Status.Error.Error01.%X13 )
   END_RUNG
   RUNG wire#powerrail
      Contact( #SS_Warning.Res_0_6 )
      Coil( #TS_Status.Error.Error01.%X14 )
   END_RUNG
   RUNG wire#powerrail
      Contact( #SS_Warning.Res_0_7 )
      Coil( #TS_Status.Error.Error01.%X15 )
   END_RUNG
   // the same network as SCL:
   #TS_Status.Error.Error01.%X8 := #SS_Warning.LimSpd;
   #TS_Status.Error.Error01.%X9 := #SS_Warning.NoTaskExec;
   #TS_Status.Error.Error01.%X10 := #SS_Warning.NotOnPath;
   #TS_Status.Error.Error01.%X11 := #SS_Warning.Res_0_3;
   #TS_Status.Error.Error01.%X12 := #SS_Warning.Res_0_4;
   #TS_Status.Error.Error01.%X13 := #SS_Warning.Res_0_5;
   #TS_Status.Error.Error01.%X14 := #SS_Warning.Res_0_6;
   #TS_Status.Error.Error01.%X15 := #SS_Warning.Res_0_7;
END_REGION

REGION Network 44: Copy temporary variables to output variables
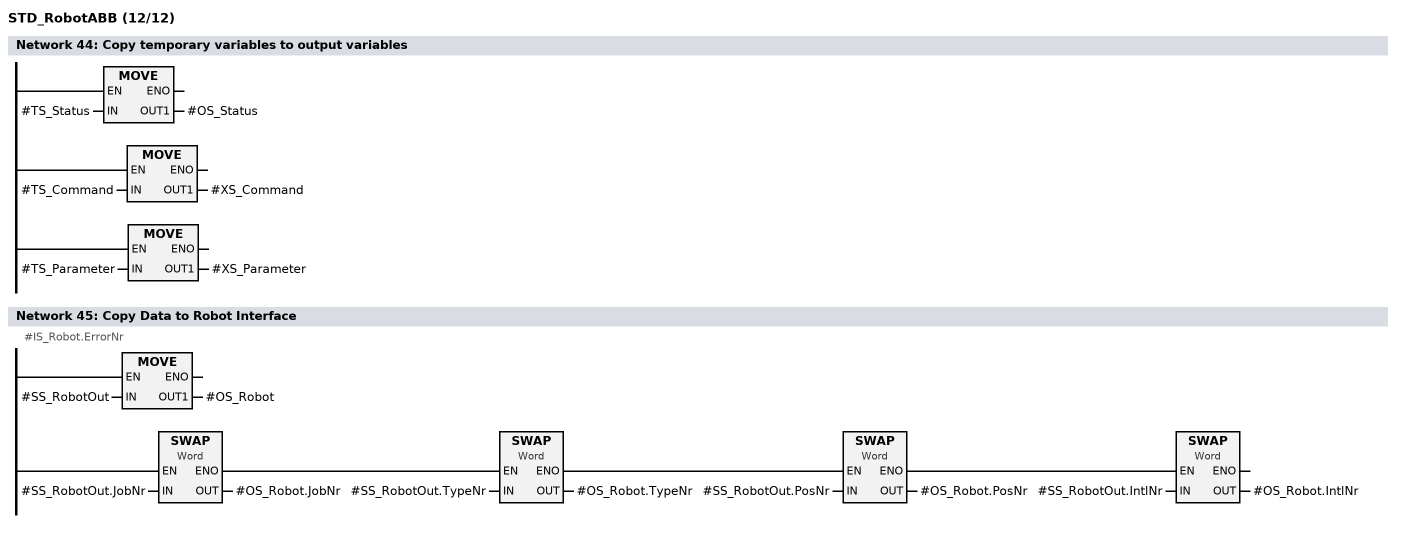
   RUNG wire#powerrail
      { S7_GenerateENO := "TRUE" } Move(in := #TS_Status, out1 => #OS_Status)
   END_RUNG
   RUNG wire#powerrail
      { S7_GenerateENO := "TRUE" } Move(in := #TS_Command, out1 => #XS_Command)
   END_RUNG
   RUNG wire#powerrail
      { S7_GenerateENO := "TRUE" } Move(in := #TS_Parameter, out1 => #XS_Parameter)
   END_RUNG
   // the same network as SCL:
   #OS_Status := #TS_Status;
   #XS_Command := #TS_Command;
   #XS_Parameter := #TS_Parameter;
END_REGION

REGION Network 45: Copy Data to Robot Interface
   // #IS_Robot.ErrorNr
   #OS_Robot := #SS_RobotOut;
   #OS_Robot.JobNr := SWAP(#SS_RobotOut.JobNr);
   #OS_Robot.TypeNr := SWAP(#SS_RobotOut.TypeNr);
   #OS_Robot.PosNr := SWAP(#SS_RobotOut.PosNr);
   #OS_Robot.IntlNr := SWAP(#SS_RobotOut.IntlNr);
END_REGION
END_FUNCTION_BLOCK
